// Timer/XPULSE
(*Ist x_Ein auf true, wird x_Aus auf true gesetzt mit der eingegebenen Ablaufzeit, unabhängig ob x_Ein früher abfällt,
als die eingegebene Ablaufzeit.
*)
FUNCTION_BLOCK XPULSE
(*
Versionsverlauf: 
Version		|Autor	|Bemerkung
------------------------------------------------------------------------------------------------------------ 
17.05.00	|KuzR	|erste Freigabe 
17.08.00	|LeaF	|Freigabe

*)
VAR_INPUT
	x_Ein:BOOL;//Eingang
END_VAR
VAR_INPUT PERSISTENT
	t_Abl:Timestruct := (wSecond := 5);//Eingegebene Ablaufzeit	
END_VAR
VAR_OUTPUT
	x_Aus:BOOL;//Digitaler Ausgang
	t_ET:Timestruct;//Ausgang Ablaufzeit
END_VAR	
VAR
	Ein:tp;
	t_PtZeit:TIME;
	Timestruct_to_Time:Timestruct_to_Time;
	Time_to_Timestruct: Time_to_Timestruct;	
END_VAR

//Wenn Eingang True, dann läuft eingestellte Zeit ab	
	Timestruct_to_Time(t_Ein:=t_Abl , t_Aus=>t_PtZeit );
	Ein(IN:= x_Ein, PT:= t_PtZeit, Q=> x_Aus);

//Ausgabe Ablaufzeit im timestruct
	Time_to_Timestruct(t_Ein:= Ein.ET, t_Aus=> t_ET);

END_FUNCTION_BLOCK

// Uhren/ABS_Bool
(*Anti Blockiersystem für BOOL Aktoren. Wird der Aktor während der eingestellten Zeit nicht bewegt so wird dieser für eine bestimmte Dauer eingeschalten.
*)
FUNCTION_BLOCK ABS_Bool
(*
Versionsverlauf: 
Version		|Autor	|Bemerkung
------------------------------------------------------------------------------------------------------------ 
17.06.00	|Shgb	|erste Freigabe 

*)
VAR_INPUT
	x_Ein:BOOL;//Eingang
END_VAR
VAR_INPUT PERSISTENT
	t_Einschaltzeitpunkt:timestruct := (wDayOfWeek := 1, wHour := 9) ;//Wochentag mit Uhrzeit wann der Ausgang geschalten wird
	t_Dauer:timestruct := (wMinute := 2);//Dauer des Force Zycklus
END_VAR
VAR_OUTPUT
	x_Aus:BOOL;//Ausgang
END_VAR
VAR
	TOF:TOF;
	Dauer:Timestruct_to_Time;
	x_Bewegt: BOOL;
	x_Flanke: BOOL;
END_VAR

// Einschalten jede Woche, eingestellte Zeit
	IF  Globale_Uhr.systemtimestruct.wDayOfWeek = t_Einschaltzeitpunkt.wDayOfWeek  AND
		Globale_Uhr.systemtimestruct.wHour = t_Einschaltzeitpunkt.wHour AND
		Globale_Uhr.systemtimestruct.wMinute = t_Einschaltzeitpunkt.wMinute THEN
		IF NOT x_Bewegt AND NOT x_Flanke THEN
			TOF.IN:=TRUE;
		ELSE
			x_Bewegt:=FALSE;
		END_IF
		x_Flanke:=TRUE;
	ELSE
		x_Flanke:=FALSE;
	END_IF
	
//Sobald Bewegt wurde Bit setzen
	IF x_Ein THEN
		x_Bewegt:=TRUE;
	END_IF

//Timestruct to Time
	Dauer(t_Ein:=t_Dauer);
	TOF(PT:=Dauer.t_Aus);
	TOF.IN:=FALSE;

//Ausgang setzen
	x_Aus:=x_Ein OR tof.Q;

END_FUNCTION_BLOCK

// Uhren/ABS_Int
(*Anti Blockiersystem für INT Aktoren. Der Aktor wir nach Ablauf der eingestellten Zeit auf den i_Force Wert bewegt und bleibt währen der Dauer auf diesem Wert.
*)
FUNCTION_BLOCK ABS_Int
(*
Versionsverlauf: 
Version		|Autor	|Bemerkung
------------------------------------------------------------------------------------------------------------ 
17.06.00	|Shgb	|erste Freigabe 

*)
VAR_INPUT
	i_Ein:int;//Eingang
END_VAR
VAR_INPUT PERSISTENT 
	t_Einschaltzeitpunkt:timestruct := (wDay := 7);//Zeit zwischen den einzelnen Force Zycklen
	t_Dauer:timestruct := (wMinute := 2);//Dauer des Force Zycklus
END_VAR
VAR_OUTPUT
	i_Aus:INT;//Ausgang
END_VAR
VAR
	TOF: TOF;
	Dauer: Timestruct_to_Time;
	x_Bewegt: BOOL;
	i_Speicher: INT;
	x_Flanke: BOOL;
END_VAR

// Einschalten jede Woche, eingestellte Zeit
	IF  Globale_Uhr.systemtimestruct.wDayOfWeek = t_Einschaltzeitpunkt.wDayOfWeek  AND
		Globale_Uhr.systemtimestruct.wHour = t_Einschaltzeitpunkt.wHour AND
		Globale_Uhr.systemtimestruct.wMinute = t_Einschaltzeitpunkt.wMinute THEN
		IF NOT x_Bewegt AND NOT x_Flanke THEN
			TOF.IN:=TRUE;
		ELSE
			x_Bewegt:=FALSE;
			i_Speicher:=i_Ein;
		END_IF
		x_Flanke:=TRUE;
	ELSE
		x_Flanke:=FALSE;
	END_IF
	
//Sobald Bewegt wurde Bit setzen
	IF i_Ein >= i_Speicher+10 OR i_Ein <= i_Speicher-10 THEN
		x_Bewegt:=TRUE;
	END_IF

//Timestruct to Time
	Dauer(t_Ein:=t_Dauer);
	TOF(PT:=Dauer.t_Aus);
	TOF.IN:=FALSE;

//Ausgang setzen
	IF tof.Q THEN
		i_Aus:=1000-i_Ein;	
	ELSE
		i_Aus:=i_Ein;
	END_IF;

END_FUNCTION_BLOCK

// Uhren/ABS_Real
(*Anti Blockiersystem für REAL Aktoren. Der Aktor wir nach Ablauf der eingestellten Zeit auf den f_Force Wert bewegt und bleibt währen der Dauer auf diesem Wert.
*)
FUNCTION_BLOCK ABS_Real
(*
Versionsverlauf: 
Version		|Autor	|Bemerkung
------------------------------------------------------------------------------------------------------------ 
17.06.00	|Shgb	|erste Freigabe 

*)
VAR_INPUT
	f_Ein:real;//Eingang
END_VAR
VAR_INPUT PERSISTENT 
	t_Einschaltzeitpunkt:timestruct := (wDay := 7);//Zeit zwischen den einzelnen Force Zycklen
	t_Dauer:timestruct := (wMinute := 2);//Dauer des Force Zycklus
END_VAR
VAR_OUTPUT
	f_Aus:REAL;//Ausgang
END_VAR
VAR
	TOF: TOF;
	Dauer: Timestruct_to_Time;
	x_Bewegt: BOOL;
	f_Speicher: REAL;

	x_Flanke: BOOL;
END_VAR

// Einschalten jede Woche, eingestellte Zeit
	IF  Globale_Uhr.systemtimestruct.wDayOfWeek = t_Einschaltzeitpunkt.wDayOfWeek  AND
		Globale_Uhr.systemtimestruct.wHour = t_Einschaltzeitpunkt.wHour AND
		Globale_Uhr.systemtimestruct.wMinute = t_Einschaltzeitpunkt.wMinute THEN
		IF NOT x_Bewegt AND NOT x_Flanke THEN
			TOF.IN:=TRUE;
		ELSE
			x_Bewegt:=FALSE;
			f_Speicher:=f_Ein;
		END_IF
		x_Flanke:=TRUE;
	ELSE
		x_Flanke:=FALSE;
	END_IF
	
//Sobald Bewegt wurde Bit setzen
	IF f_Ein >= f_Speicher+10 OR f_Ein <= f_Speicher-10 THEN
		x_Bewegt:=TRUE;
	END_IF

//Timestruct to Time
	Dauer(t_Ein:=t_Dauer);
	TOF(PT:=Dauer.t_Aus);
	TOF.IN:=FALSE;

//Ausgang setzen
	IF tof.Q THEN
		f_Aus:=100-f_Ein;	
	ELSE
		f_Aus:=f_Ein;
	END_IF;

END_FUNCTION_BLOCK

// Uhren/CLK_D
(*Uhr mit Tagesprogramm. Einschaltzeit => t_Ein.wHour, t_ein.wMinute und Ausschaltzeit => t_Aus.wHour und t_Aus.wMinute. Eingabe im Timestruct Format.
Vergleicht Ein- und Ausschaltzeit mit der Globalen_Uhr(Globale Variable)
*)
FUNCTION_BLOCK CLK_D
(*
Versionsverlauf: 
Version		|Autor	|Bemerkung
------------------------------------------------------------------------------------------------------------ 
17.06.00	|KuzR	|erste Freigabe 
17.08.00	|LeaF	|Freigabe

*)
VAR_INPUT Persistent
	t_Ein:timestruct;//Eingabe Einschaltzeit 
	t_Aus:timestruct;//Eingabe Ausschaltzeit 
END_VAR
VAR_OUTPUT
	x_Aus:BOOL;//Digitaler Ausgang		 
END_VAR
VAR
END_VAR

//schaltet jeden Tag ein, eingestell e Zeit  
	IF Globale_Uhr.systemtimestruct.wHour = t_Ein.wHour AND
 	   Globale_Uhr.systemtimestruct.wMinute >= t_Ein.wMinute THEN
			x_Aus:= TRUE;
	END_IF
				
//schaltet jeden Tag wieder aus, eingestellte Zeit			
	IF 	Globale_Uhr.systemtimestruct.wHour = t_Aus.wHour AND
		Globale_Uhr.systemtimestruct.wMinute >= t_Aus.wMinute THEN
			x_Aus:= FALSE;
	END_IF

END_FUNCTION_BLOCK

// Uhren/CLK_I
(*Uhr mit einem Impuls pro Tag. Einschaltzeit => t_Ein.wHour, t_ein.wMinute und Impulszeit => t_Imp.w.Second Eingabe im Timestruct Format. Vergleicht Einschaltzeit 
mit der Globalen_Uhr(Globale Variable)
*)
FUNCTION_BLOCK CLK_I
(*
Versionsverlauf: 
Version		|Autor	|Bemerkung
------------------------------------------------------------------------------------------------------------ 
17.06.00	|KuzR	|erste Freigabe 
17.08.00	|LeaF	|Freigabe

*)
VAR_INPUT Persistent
 	t_Ein:timestruct;//Eingabe Einschaltzeit 
	t_Imp:timestruct;//Eingabe Impulszeit
END_VAR
VAR_OUTPUT
	x_Aus:BOOL;//Digitaler Ausgang			 
END_VAR
VAR	
	impuls:tp;
	x_Zeit_groesser:BOOL;   
	t_ptImpuls: TIME;
	Timestruct_to_Time: Timestruct_to_Time;
END_VAR

//schaltet jeden Tag ein, eingestellte Zeit
	IF Globale_Uhr.systemtimestruct.wHour = t_Ein.wHour AND
 	   Globale_Uhr.systemtimestruct.wMinute >= t_Ein.wMinute THEN
			x_Zeit_groesser	:=TRUE;		
	ELSE
			x_Zeit_groesser :=  FALSE;
	END_IF
				
//Impulsdauer
	Timestruct_to_Time(t_Ein:=t_Imp , t_Aus=>t_ptImpuls );
	impuls(in:=x_Zeit_groesser, pt:=t_ptImpuls);
		x_Aus:= impuls.Q;
		x_Zeit_groesser:= x_Aus;

END_FUNCTION_BLOCK

// Uhren/CLK_M
(*Uhr mit Monatsprogramm. Schaltet 1mal im Monat für eine einstellbare Zeit.  Einschaltzeit => t_Ein.wDay, t_Ein.wHour, t_ein.wMinute
und Ausschaltzeit => t_Ein.wDay, t_Ein.wHour, t_ein.wMinute.
Eingabe im Timestruct Format. Vergleicht Ein- und Ausschaltzeit mit der Globalen_Uhr(Globale Variable)
*)
FUNCTION_BLOCK CLK_M
(*
Versionsverlauf: 
Version		|Autor	|Bemerkung
------------------------------------------------------------------------------------------------------------ 
17.06.00	|KuzR	|erste Freigabe 
17.08.00	|LeaF	|Freigabe

*)
VAR_INPUT Persistent
	    t_Ein:timestruct;//Eingabe Einschaltzeit 
		t_Aus:timestruct;//Eingabe Ausschaltzeit 	
END_VAR
VAR_OUTPUT
		x_Aus:BOOL;	 
END_VAR
VAR
	
		
	
	
	

		
	
	
END_VAR

// Einschalten einmal im Monat, Tag und Zeit
	IF  Globale_Uhr.systemtimestruct.wDay = t_Ein.wDay  AND
		Globale_Uhr.systemtimestruct.wHour = t_Ein.wHour AND
		Globale_Uhr.systemtimestruct.wMinute >= t_Ein.wMinute THEN
			x_Aus:= TRUE;
	END_IF
	
// Ausschalten einmal im Monat, Tag und Zeit
	IF  Globale_Uhr.systemtimestruct.wDay = t_Aus.wDay  AND
		Globale_Uhr.systemtimestruct.wHour = t_Aus.wHour AND
		Globale_Uhr.systemtimestruct.wMinute >= t_Aus.wMinute THEN
			x_Aus:= FALSE;
	END_IF

END_FUNCTION_BLOCK

// Uhren/CLK_W
(*Uhr mit Wochernprogramm. Schaltet 1 mal in der Woche für eine einstellbare Zeit.  Einschaltzeit => t_Ein.wDayofWeek, t_Ein.wHour, t_ein.wMinute
und Ausschaltzeit => t_Ein.wDayofWeek, t_Ein.wHour, t_ein.wMinute.
Eingabe im Timestruct Format. Vergleicht Ein- und Ausschaltzeit mit der Globalen_Uhr(Globale Variable)
*)
FUNCTION_BLOCK CLK_W
(*
Versionsverlauf: 
Version		|Autor	|Bemerkung
------------------------------------------------------------------------------------------------------------ 
17.06.00	|KuzR	|erste Freigabe 
17.08.00	|LeaF	|Freigabe

*)
VAR_INPUT Persistent
	t_Ein:timestruct;//Eingabe Einschaltzeit 
	t_Aus:timestruct;//Eingabe Ausschaltzeit
END_VAR
VAR_OUTPUT
	x_Aus:BOOL;//Digitaler Ausgang 
END_VAR

// Einschalten jede Woche, eingestellte Zeit
	IF  Globale_Uhr.systemtimestruct.wDayOfWeek = t_Ein.wDayOfWeek  AND
		Globale_Uhr.systemtimestruct.wHour = t_Ein.wHour AND
		Globale_Uhr.systemtimestruct.wMinute >= t_Ein.wMinute THEN
			x_Aus:= TRUE;
	END_IF
// Ausschalten, eingestellte Zeit
	IF  Globale_Uhr.systemtimestruct.wDayOfWeek = t_Aus.wDayOfWeek  AND
		Globale_Uhr.systemtimestruct.wHour = t_Aus.wHour AND
		Globale_Uhr.systemtimestruct.wMinute >= t_Aus.wMinute THEN
			x_Aus:= FALSE;
	END_IF

END_FUNCTION_BLOCK

// Uhren/CLK_W7
(*Uhr mit Wochenprogramm für jeden Wochentag. Schaltet 1 mal im Tag für eine einstellbare Zeit, jeden Wochentag einzeln wählbar.
Einschaltzeit => t_Ein.wHour, t_ein.wMinute
und Ausschaltzeit => t_Ein.wHour, t_ein.wMinute
Eingabe im Timestruct Format. Vergleicht Ein- und Ausschaltzeit mit der Globalen_Uhr(Globale Variable)
*)
FUNCTION_BLOCK CLK_W7
(*
Versionsverlauf: 
Version		|Autor	|Bemerkung
------------------------------------------------------------------------------------------------------------ 
17.06.00	|KuzR	|erste Freigabe 
17.08.00	|LeaF	|Freigabe

*)
VAR_INPUT Persistent	   	
		t_Ein_Mo:timestruct;//Eingabe Einschaltzeit Montag
		t_Aus_Mo:timestruct;//Eingabe Ausschaltzeit Montag
 		t_Ein_Di:timestruct;//Eingabe Einschaltzeit Dienstag
		t_Aus_Di:timestruct;//Eingabe Ausschaltzeit Dienstag
		t_Ein_Mi:timestruct;//Eingabe Einschaltzeit Mittwoch
		t_Aus_Mi:timestruct;//Eingabe Ausschaltzeit Mittwoch
		t_Ein_Do:timestruct;//Eingabe Einschaltzeit Donnerstag
		t_Aus_Do:timestruct;//Eingabe Ausschaltzeit Donnerstag
		t_Ein_Fr:timestruct;//Eingabe Einschaltzeit Freitag
		t_Aus_Fr:timestruct;//Eingabe Ausschaltzeit Freitag
		t_Ein_Sa:timestruct;//Eingabe Einschaltzeit Samstag
		t_Aus_Sa:timestruct;//Eingabe Ausschaltzeit Samstag
		t_Ein_So:timestruct;//Eingabe Einschaltzeit Sonntag
		t_Aus_So:timestruct;//Eingabe Ausschaltzeit Sonntag
END_VAR
VAR_OUTPUT
		x_Aus:BOOL;//Digitaler Ausgang	 
END_VAR
VAR
END_VAR

//Montag einschalten
	IF  Globale_Uhr.systemtimestruct.wDayOfWeek = 1  AND
		Globale_Uhr.systemtimestruct.wHour = t_Ein_Mo.wHour AND
		Globale_Uhr.systemtimestruct.wMinute >= t_Ein_Mo.wMinute THEN
			x_Aus:= TRUE;
			END_IF
//Montag ausschalten	
	IF  Globale_Uhr.systemtimestruct.wDayOfWeek = 1  AND
		Globale_Uhr.systemtimestruct.wHour = t_Aus_MO.wHour AND
		Globale_Uhr.systemtimestruct.wMinute >= t_Aus_MO.wMinute THEN
			x_Aus:= FALSE;
			END_IF
//Dienstag einschalten
	IF  Globale_Uhr.systemtimestruct.wDayOfWeek = 2  AND
		Globale_Uhr.systemtimestruct.wHour = t_Ein_Di.wHour AND
		Globale_Uhr.systemtimestruct.wMinute >= t_Ein_Di.wMinute THEN
			x_Aus:= TRUE;
			END_IF
//Dienstag ausschalten	
	IF  Globale_Uhr.systemtimestruct.wDayOfWeek = 2  AND
		Globale_Uhr.systemtimestruct.wHour = t_Aus_Di.wHour AND
		Globale_Uhr.systemtimestruct.wMinute >= t_Aus_Di.wMinute THEN
			x_Aus:= FALSE;
			END_IF
//Mittwoch einschalten
	IF  Globale_Uhr.systemtimestruct.wDayOfWeek = 3  AND
		Globale_Uhr.systemtimestruct.wHour = t_Ein_Mi.wHour AND
		Globale_Uhr.systemtimestruct.wMinute >= t_Ein_Mi.wMinute THEN
			x_Aus:= TRUE;
			END_IF
//Mittwoch ausschalten	
	IF  Globale_Uhr.systemtimestruct.wDayOfWeek = 3  AND
		Globale_Uhr.systemtimestruct.wHour = t_Aus_Mi.wHour AND
		Globale_Uhr.systemtimestruct.wMinute >= t_Aus_Mi.wMinute THEN
			x_Aus:= FALSE;
			END_IF		
//Donnerstag einschalten
	IF  Globale_Uhr.systemtimestruct.wDayOfWeek = 4  AND
		Globale_Uhr.systemtimestruct.wHour = t_Ein_Do.wHour AND
		Globale_Uhr.systemtimestruct.wMinute >= t_Ein_Do.wMinute THEN
			x_Aus:= TRUE;
			END_IF
//Donnerstag ausschalten	
	IF  Globale_Uhr.systemtimestruct.wDayOfWeek = 4  AND
		Globale_Uhr.systemtimestruct.wHour = t_Aus_Do.wHour AND
		Globale_Uhr.systemtimestruct.wMinute >= t_Aus_Do.wMinute THEN
			x_Aus:= FALSE;
			END_IF

//Freitag einschalten
	IF  Globale_Uhr.systemtimestruct.wDayOfWeek = 5  AND
		Globale_Uhr.systemtimestruct.wHour = t_Ein_Fr.wHour AND
		Globale_Uhr.systemtimestruct.wMinute >= t_Ein_Fr.wMinute THEN
			x_Aus:= TRUE;
			END_IF
//Freitag ausschalten	
	IF  Globale_Uhr.systemtimestruct.wDayOfWeek = 5  AND
		Globale_Uhr.systemtimestruct.wHour = t_Aus_Fr.wHour AND
		Globale_Uhr.systemtimestruct.wMinute >= t_Aus_Fr.wMinute THEN
			x_Aus:= FALSE;
			END_IF		
//Samstag einschalten
	IF  Globale_Uhr.systemtimestruct.wDayOfWeek = 6  AND
		Globale_Uhr.systemtimestruct.wHour = t_Ein_Sa.wHour AND
		Globale_Uhr.systemtimestruct.wMinute >= t_Ein_Sa.wMinute THEN
			x_Aus:= TRUE;
			END_IF
//Samstag ausschalten	
	IF  Globale_Uhr.systemtimestruct.wDayOfWeek = 6  AND
		Globale_Uhr.systemtimestruct.wHour = t_Aus_Sa.wHour AND
		Globale_Uhr.systemtimestruct.wMinute >= t_Aus_Sa.wMinute THEN
			x_Aus:= FALSE;
			END_IF	
//Sonntag einschalten
	IF  Globale_Uhr.systemtimestruct.wDayOfWeek = 0  AND
		Globale_Uhr.systemtimestruct.wHour = t_Ein_So.wHour AND
		Globale_Uhr.systemtimestruct.wMinute >= t_Ein_So.wMinute THEN
			x_Aus:= TRUE;
			END_IF
//Sonntag ausschalten	
	IF  Globale_Uhr.systemtimestruct.wDayOfWeek = 0  AND
		Globale_Uhr.systemtimestruct.wHour = t_Aus_So.wHour AND
		Globale_Uhr.systemtimestruct.wMinute >= t_Aus_So.wMinute THEN
			x_Aus:= FALSE;
			END_IF

END_FUNCTION_BLOCK

// Uhren/CLK_Y
(*Uhr mit Jahresrogramm. Schaltet 1 mal im Jahr für eine einstellbare Zeit.  Einschaltzeit => t_Ein.wMonth, t_Ein.wDay, t_Ein.wHour, t_ein.wMinute
und Ausschaltzeit => t_Aus.wMonth, t_Ein.wDay, t_Ein.wHour, t_ein.wMinute.
Eingabe im Timestruct Format. Vergleicht Ein- und Ausschaltzeit mit der Globalen_Uhr(Globale Variable)
*)
FUNCTION_BLOCK CLK_Y
(*
Versionsverlauf: 
Version		|Autor	|Bemerkung
------------------------------------------------------------------------------------------------------------ 
17.06.00	|KuzR	|erste Freigabe 
17.08.00	|LeaF	|Freigabe

*)
VAR_INPUT Persistent
	t_Ein:timestruct;//Eingabe Einschaltzeit
	t_Aus:timestruct;//Eingabe Ausschaltzeit	

END_VAR
VAR_OUTPUT
	x_Aus:BOOL;			 
END_VAR
VAR
END_VAR

// Einschalten einmal im Jahr, Zeit, Tagnummer und Monat
	IF Globale_Uhr.systemtimestruct.wMonth = t_Ein.wMonth AND
 	   Globale_Uhr.systemtimestruct.wDay = t_Ein.wDay AND
	   Globale_Uhr.systemtimestruct.wHour = t_Ein.wHour AND
	   Globale_Uhr.systemtimestruct.wMinute >= t_Ein.wMinute THEN
			x_Aus:= TRUE;		
	END_IF
			
// Ausschalten Zeit, Tagnummer und Monat 	
	IF Globale_Uhr.systemtimestruct.wMonth = t_Aus.wMonth AND
 	   Globale_Uhr.systemtimestruct.wDay = t_Aus.wDay AND
	   Globale_Uhr.systemtimestruct.wHour = t_Aus.wHour AND
	   Globale_Uhr.systemtimestruct.wMinute >= t_Aus.wMinute THEN			
			x_Aus:= FALSE;
	END_IF

END_FUNCTION_BLOCK

// Uhren/FerienPRG
(*FB Ferienprogramm, Wenn FB aktiviert und die Schaltuhr aktiv ist, schaltet die Freigabe x_BM und der Sollwert Eingang wird auf
den Ausgang geschrieben. Es muss nur die Ausschaltzeit eingegeben werden t_Aus.wMonth, => t_Aus.wDay, t_Aus.wHour, t_Aus.wMinute.
Sobald die Zeit abgelaufen ist, wird der Sollwert Ausgang auf 0 gesetzt und der Ausgang x_BM wird auf false gesetzt.
*)
FUNCTION_BLOCK FerienPRG
(*
Versionsverlauf: 
Version		|Autor	|Bemerkung
------------------------------------------------------------------------------------------------------------ 
17.07.00	|KuzR	|erste Freigabe 
17.08.00	|LeaF	|Freigabe

*)
VAR_INPUT PERSISTENT
	x_Akt:BOOL;//Aktivierung
	t_Aus:TIMESTRUCT;//Ausschaltzeit
	f_SW_fix:REAL;//Sollwert
END_VAR
VAR_OUTPUT
	x_BM:BOOL;//Freigabe
	f_SW:REAL;//Sollwert
	t_Restzeit:timestruct;//Anzeige Restzeit
END_VAR
VAR
	ein: BOOL;
	x_Aus_Uhr:BOOL;
	x_ein:BOOL;
	t_Restzeit1:TIME;
	t_Ausschalt: TIME;
	t_Global:TIME;
	CLK_M: CLK_M;
	Timestruct_to_Time: Timestruct_to_Time;
	Time_to_Timestruct: Time_to_Timestruct;
	SWITCH_REAL: SWITCH_REAL;
	
	CLK_Y: CLK_Y;
END_VAR

//Kommentar

//Monatsuhr, Zeiteingabe im Timestruct
		CLK_Y(t_Ein:= Globale_Uhr.systemtimestruct, t_Aus:=t_Aus , x_Aus=>x_Aus_Uhr );
//Freigabe schalten
 		x_BM:= x_Akt AND x_Aus_Uhr;

//Timestruct to time
		Timestruct_to_Time(t_Ein:=t_Aus , t_Aus=>t_Ausschalt );
		Timestruct_to_Time(t_Ein:=Globale_Uhr.systemtimestruct , t_Aus=>t_Global);	
			
//Restzeit berechnen im Time Format
		t_Restzeit1:=t_Ausschalt-t_Global;
	IF t_Ausschalt < t_Global THEN
		t_Restzeit1:=T#0S;
	END_IF
	
//Time to timestruct
	Time_to_Timestruct(t_Ein:= t_Restzeit1, t_Aus=> t_Restzeit);

//Sollwert in den Ausgang schreiben	
	SWITCH_REAL(x_Ein:=x_BM , f_Ein_1:=0 , f_Ein_2:=f_SW_fix , f_Aus=>f_SW );
		
	IF NOT x_Aus_Uhr THEN
		x_Akt:=FALSE;
	END_IF

END_FUNCTION_BLOCK

// Verdichter/Einsatzgrenzen_Normal
(*Überwacht die Einsatzgrenzen der Kompressoren und gibt mit einem BOOL an ob diese sich noch in den Einsatzgrenzen befinden. Ein Toleranzband kann zusätzlich mit einer Zeit bestimmt werden.
Verlässt der Kompressor die Einsatzgrenzen ober wird zu lange im Toleranzband betrieben so wird das Ausgangsbool auf FALSE gesetzt. Für weitere Infos siehe Beschrieb im FB.
*)
FUNCTION_BLOCK Einsatzgrenzen_Normal
(*
Versionsverlauf: 
Version		|Autor	|Bemerkung
------------------------------------------------------------------------------------------------------------ 
17.06.00	|Shgb	|erste Freigabe 
17.06.01	|ShgB	|von Integer auf Real geändert
17.06.02	|ShgB	|Von Time auf Timestruct geändert
17.07.00	|ShgB	|MOP Berechnung angepasst

		  F	_____________5__________ E
		  /							\ 4
	  6	/							 \ D
	  /								 | 3
  G /								 | C
	|								/  
	|							  /
  7 |							/ 2
	|_________________________/
	A			1			  B
*)
VAR_INPUT 
	f_Verd:REAL;//Aktuelle Verdampfungstemperatur
	f_Kond:REAL;//Aktuelle Kondensationstemperatur
	x_Betriebsmeldung: BOOL;//Sobald die Betriebsmeldung kommt wird die Auswertung um die eingestellte Zeit verzögert aktiv
	x_SW_Reset:BOOL;//Setzt die Standardwerte für den Kompressorty zurück
	dut_Kompressortyp:SW_Einsatzgrenzen:=SW_ALZ.Bitzer_Scroll_R410a;//Kompressortyp als DUT Angabe Standard Bitzer Scroll 410a
END_VAR
VAR_INPUT PERSISTENT
	f_MinVerd:REAL;//Minimale Verdampfungstemperatur Linie 7
	f_MaxVerd:REAL;//Maximale Verdampfungstemperatur Linie 3
	f_MinKond:REAL;//Minimale Kondensationstemperatur Punkt A
	f_MaxKond:REAL;//Maximale Kondensationstemperatur Linie 5
	f_BVerd:REAL;//Verdampfungstemperatur beim Punkt B
	f_BKond:REAL;//Kondensationstemperatur beim Punkt B
	f_CKond:REAL;//Kondensationstemperatur beim Punkt C
	f_DKond:REAL;//Kondensationstemperatur beim Punkt D
	f_EVerd:REAL;//Verdampfungstemperatur beim Punkt E
	f_FVerd:REAL;//Verdampfungstemperatur beim Punkt F
	f_GKond:REAL;//Kondensationstemperatur beim Punkt G
	f_Toleranz:REAL:=1;//Breite des Toleranzbandes in °C
	t_Toleranz:timestruct := (wMinute := 5);//Zeit die der Kompressor im Toleranzband sein darf
	f_GUI_Zoom:REAL;//Zoomfaktor für das Vergrössern der Grafik
	i_GUI_VersatzX:INT;//Versatz der Grafik in X Richtung (Verdampfung)
	i_GUI_VersatzY:INT;//Versatz der Grafik in Y Richtung (Kondensation)
END_VAR
VAR_OUTPUT
	f_ActMinKond:REAL;//Aktuelle mindest Kondensation laut Einsatzgrenzendiagramm
	f_ActMaxKond:REAL;//Aktuelle maximale Kondensation laut Einsatzgrenzendiagramm
	f_ActMinVerd:REAL;//Aktuelle mindest Verdampfung laut Einsatgrenzendiagramm
	f_ActMaxVerd:REAL;//Aktuelle maximale Verdampfung laut Einsatzgrenzendiagramm
	x_Aus:BOOL;//Befindet sich der Kompressor in den Einsatzgrenzen
	x_BM_ND:BOOL;//Kompressor befindet sich im Toleranzband auf der Niederdruckseite
	x_AL_ND:BOOL;//Kompressor ist ausserhalb der Einsatzgrenzen auf der Niederdruckseite
	x_BM_HD:BOOL;//Kompressor befindet sich im Toleranzband auf der Hochdruckseite
	x_AL_HD:BOOL;//Kompressor ist ausserhalb der Einsatzgrenzen auf der Hochdruckseite
	x_BM_MOP: BOOL;//Kompressor befindet sich im Toleranzband vor dem MOP Alarm
	x_AL_MOP: BOOL;//MOP wurde überschritten
END_VAR
VAR
	Timer: TON;
	x_Timer:BOOL;
	Maximum: Maximum;
	Linie1_Verd: Converter2Punkt;
	Linie1_Kond: Converter2Punkt;
	Linie2_Verd: Converter2Punkt;
	Linie2_Kond: Converter2Punkt;
	Linie4_Kond: Converter2Punkt;
	Linie4_Verd: Converter2Punkt;
	Linie6_Verd: Converter2Punkt;
	Linie6_Kond: Converter2Punkt;
	Minimum: Minimun;
	t_Temp: TIME;
	Timestruct_to_Time:Timestruct_to_Time;
	FB_MIN_KD: maximum;
	FB_MIN_VD: maximum;
	FB_MAX_KD: Minimun;
	FB_MAX_VD: Minimun;
	Betriebsmeldung:Ton;
END_VAR
VAR PERSISTENT
	x_Laden:BOOL;//Variable ist beim ersten aufstarten False und lädt somit die eingestellten Daten
END_VAR
VAR//Variablen für Grafik
	f_GUI_Verd:REAL;//Aktuelle Verdampfungstemperatur
	f_GUI_Kond:REAL;//Aktuelle Kondensationstemperatur
	f_GUI_MinVerd:REAL;//Minimale Verdampfungstemperatur Linie 7
	f_GUI_MaxVerd:REAL;//Maximale Verdampfungstemperatur Linie 3
	f_GUI_MinKond:REAL;//Minimale Kondensationstemperatur Punkt A
	f_GUI_MaxKond:REAL;//Maximale Kondensationstemperatur Linie 5
	f_GUI_BVerd:REAL;//Verdampfungstemperatur beim Punkt B
	f_GUI_BKond:REAL;//Kondensationstemperatur beim Punkt B
	f_GUI_CKond:REAL;//Kondensationstemperatur beim Punkt C
	f_GUI_DKond:REAL;//Kondensationstemperatur beim Punkt D
	f_GUI_EVerd:REAL;//Verdampfungstemperatur beim Punkt E
	f_GUI_FVerd:REAL;//Verdampfungstemperatur beim Punkt F
	f_GUI_GKond:REAL;//Kondensationstemperatur beim Punkt G
END_VAR

//Linienberechnungen
	//Linie 1
		Linie1_Verd(
			f_Ein:= f_Verd, 
			f_Ein_Min:= f_MinVerd, 
			f_Ein_Max:= f_BVerd, 
			f_Aus_Min:= f_MinKond, 
			f_Aus_Max:= f_BKond);
			
		Linie1_Kond(
			f_Ein:= f_Kond, 
			f_Ein_Min:= f_MinKond, 
			f_Ein_Max:= f_BKond, 
			f_Aus_Min:= f_MinVerd, 
			f_Aus_Max:= f_BVerd);
			
	//Linie 2
		Linie2_Verd(
			f_Ein:= f_Verd, 
			f_Ein_Min:= f_BVerd, 
			f_Ein_Max:= f_MaxVerd, 
			f_Aus_Min:= f_BKond, 
			f_Aus_Max:= f_CKond);
			
		Linie2_Kond(
			f_Ein:= f_Kond, 
			f_Ein_Min:= f_BVerd, 
			f_Ein_Max:= f_MaxVerd, 
			f_Aus_Min:= f_BKond, 
			f_Aus_Max:= f_CKond);
			
	//Linie 4
		Linie4_Kond(
			f_Ein:= f_Kond, 
			f_Ein_Min:= f_MaxKond, 
			f_Ein_Max:= f_DKond, 
			f_Aus_Min:= f_EVerd, 
			f_Aus_Max:= f_MaxVerd);
			
		Linie4_Verd(
			f_Ein:= f_Verd, 
			f_Ein_Min:= f_EVerd, 
			f_Ein_Max:= f_MaxVerd, 
			f_Aus_Min:= f_MaxKond, 
			f_Aus_Max:= f_DKond);
			
	//Linie 6
		Linie6_Verd(
			f_Ein:= f_Verd, 
			f_Ein_Min:= f_MinVerd, 
			f_Ein_Max:= f_FVerd, 
			f_Aus_Min:= f_GKond, 
			f_Aus_Max:= f_MaxKond);
				
		Linie6_Kond(
			f_Ein:= f_Kond, 
			f_Ein_Min:= f_GKond, 
			f_Ein_Max:= f_MaxKond, 
			f_Aus_Min:= f_MinVerd, 
			f_Aus_Max:= f_FVerd);
			
//Minimale Kondensationstemperatur wird durch die Linien 1,  2 und f_MinKond vom Einsatzgrenzendiagramm gegeben. Die höhere von beiden wird genommen.
	FB_MIN_KD(
		f_Ein1:= Linie1_Verd.f_Aus, 
		f_Ein2:= Linie2_Verd.f_Aus, 
		f_Ein3:= f_MinKond, 
		f_Aus=> f_ActMinKond);
			
//Maximale Kondensationstemperaturwird durch Linie 4, 6 und f_MaxKond vom Einsatzgrenzendiagramm gegeben. Die kleinere von den dreien wird genommen. Linie 5 ist f_MaxKond
	FB_MAX_KD(
		f_Ein1:=Linie4_Verd.f_Aus,
		f_Ein2:=Linie6_Verd.f_Aus,
		f_Ein3:=f_MaxKond,
		f_Aus=>f_ActMaxKond);
			
//Minimale Verdampfungstemperatur durch Linie 6 und f_MinVerd gegeben
	FB_MIN_VD(
		f_Ein1:=Linie6_Kond.f_Aus,
		f_Ein2:= f_MinVerd,
		f_Aus=>f_ActMinVerd);
				
//Maximale Verdampfungstemperatur 
	IF f_Kond <= f_BKond AND f_Kond>= f_MinKond THEN
		f_ActMaxVerd:=Linie1_Kond.f_Aus;
	ELSE
		FB_MAX_VD(
			f_Ein1:=Linie2_Kond.f_Aus,
			f_Ein2:=Linie4_Kond.f_Aus,
			f_Ein3:=f_MaxVerd,
			f_Aus=>f_ActMaxVerd);
	END_IF

//TImestruct to Time
	Timestruct_to_Time(t_Ein:=t_Toleranz);
	
//Auswertung ob in den Einsatzgrenzen mit Timer
	Betriebsmeldung(IN:=x_Betriebsmeldung,PT:=Timestruct_to_Time.t_Aus);

	Timer(IN:= f_Verd < f_ActMinVerd+f_Toleranz OR
		f_Verd > f_ActMaxVerd-f_Toleranz OR
		f_Kond < f_ActMinKond+f_Toleranz OR
		f_Kond > f_ActMaxKond-f_Toleranz, PT:= Timestruct_to_Time.t_Aus, Q=> x_Timer, ET=> );
			
	x_Aus :=NOT Betriebsmeldung.Q OR(f_Verd > f_ActMinVerd AND
		f_Verd < f_ActMaxVerd AND
		f_Kond > f_ActMinKond AND
		f_Kond < f_ActMaxKond AND
		NOT x_Timer);

//Alarme
	IF Globale_Variablen.x_Quittieren THEN
		x_AL_HD := FALSE;
		x_AL_ND := FALSE;
		x_AL_MOP:= FALSE;
	END_IF

	x_BM_ND:=f_Verd<f_ActMinVerd+f_Toleranz;
		
	IF f_Verd<f_ActMinVerd THEN
		x_AL_ND:=TRUE;
	END_IF
		
	x_BM_HD:=f_Kond>f_ActMaxKond-f_Toleranz;
		
	IF f_Kond>f_ActMaxKond THEN
		x_AL_HD:=TRUE;
	END_IF
	
	x_BM_MOP:=f_Verd>f_ActMaxVerd-f_Toleranz;
	
	IF f_Verd>f_ActMaxVerd THEN
		x_AL_MOP:=TRUE;
	END_IF
	
//Reset Sollwerte
	IF x_SW_Reset OR not x_Laden THEN
		f_MinVerd:=dut_Kompressortyp.f_SW_EG_MinVerd;
		f_MaxVerd:=dut_Kompressortyp.f_SW_EG_MaxVerd;
		f_MinKond:=dut_Kompressortyp.f_SW_EG_MinKond;
		f_MaxKond:=dut_Kompressortyp.f_SW_EG_MaxKond;
		f_BVerd:=dut_Kompressortyp.f_SW_EG_BVerd;
		f_BKond:=dut_Kompressortyp.f_SW_EG_BKond;
		f_CKond:=dut_Kompressortyp.f_SW_EG_CKond;
		f_DKond:=dut_Kompressortyp.f_SW_EG_DKond;
		f_EVerd:=dut_Kompressortyp.f_SW_EG_EVerd;
		f_FVerd:=dut_Kompressortyp.f_SW_EG_FVerd;
		f_GKond:=dut_Kompressortyp.f_SW_EG_GKond;
		x_Laden:=TRUE;
	END_IF
	
//GUI Anpassungen
	f_GUI_Verd:=f_Verd*f_GUI_Zoom+i_GUI_VersatzX;
	f_GUI_Kond:=f_Kond*f_GUI_Zoom+i_GUI_VersatzY*-1;
	f_GUI_MinVerd:=f_MinVerd*f_GUI_Zoom+i_GUI_VersatzX;
	f_GUI_MaxVerd:=f_MaxVerd*f_GUI_Zoom+i_GUI_VersatzX;
	f_GUI_MinKond:=f_MinKond*f_GUI_Zoom+i_GUI_VersatzY*-1;
	f_GUI_MaxKond:=f_MaxKond*f_GUI_Zoom+i_GUI_VersatzY*-1;
	f_GUI_BVerd:=f_BVerd*f_GUI_Zoom+i_GUI_VersatzX;
	f_GUI_BKond:=f_BKond*f_GUI_Zoom+i_GUI_VersatzY*-1;
	f_GUI_CKond:=f_CKond*f_GUI_Zoom+i_GUI_VersatzY*-1;
	f_GUI_DKond:=f_DKond*f_GUI_Zoom+i_GUI_VersatzY*-1;
	f_GUI_EVerd:=f_EVerd*f_GUI_Zoom+i_GUI_VersatzX;
	f_GUI_FVerd:=f_FVerd*f_GUI_Zoom+i_GUI_VersatzX;
	f_GUI_GKond:=f_GKond*f_GUI_Zoom+i_GUI_VersatzY*-1;

END_FUNCTION_BLOCK

// Verdichter/FIFO
(*Funktionsbaustein zum Abgleich der Betriebsstunden. Der Kompressor mit der geringeren Anzahl an Betriebsstunden wird als nächstes in Betrieb genommen. 
Beim Ausschalten werden die Kompressoren nach dem FIFO (First in frist out) Prinzip ausgeschalten.
*)
FUNCTION_BLOCK FIFO
(*
Versionsverlauf: 
Version		|Autor	|Bemerkung
------------------------------------------------------------------------------------------------------------ 
17.06.00	|Shgb	|erste Freigabe
17.07.00	|Shgb	|Bool zum Kompressorwechsel
17.08.00	|LeaF	|Freigabe

*)
VAR_INPUT
	i_Stufen:INT;//Anzahl der angeforderten Stufen
	x_En1:BOOL;//Betriebstunden von Kompressor 1
	t_Betriebsstunden1:timestruct;//Betriebstunden von Kompressor 1
	x_En2:BOOL;//Betriebstunden von Kompressor 2
	t_Betriebsstunden2:timestruct;//Betriebstunden von Kompressor 2
	x_En3:BOOL;//Betriebstunden von Kompressor 3
	t_Betriebsstunden3:timestruct;//Betriebstunden von Kompressor 3
	x_En4:BOOL;//Betriebstunden von Kompressor 4
	t_Betriebsstunden4:timestruct;//Betriebstunden von Kompressor 4
	x_En5:BOOL;//Betriebstunden von Kompressor 5
	t_Betriebsstunden5:timestruct;//Betriebstunden von Kompressor 5
	x_En6:BOOL;//Betriebstunden von Kompressor 6
	t_Betriebsstunden6:timestruct;//Betriebstunden von Kompressor 6
	x_En7:BOOL;//Betriebstunden von Kompressor 7
	t_Betriebsstunden7:timestruct;//Betriebstunden von Kompressor 7
	x_En8:BOOL;//Betriebstunden von Kompressor 8
	t_Betriebsstunden8:timestruct;//Betriebstunden von Kompressor 8
	x_Wechsel: BOOL;	// Befhel für die Umschaltung der betriebenen Kompressoren.
END_VAR
VAR_OUTPUT
	x_Aus1:BOOL;//Einschaltbefehl Kompressor 1
	x_Aus2:BOOL;//Einschaltbefehl Kompressor 2
	x_Aus3:BOOL;//Einschaltbefehl Kompressor 3
	x_Aus4:BOOL;//Einschaltbefehl Kompressor 4
	x_Aus5:BOOL;//Einschaltbefehl Kompressor 5
	x_Aus6:BOOL;//Einschaltbefehl Kompressor 6
	x_Aus7:BOOL;//Einschaltbefehl Kompressor 7
	x_Aus8:BOOL;//Einschaltbefehl Kompressor 8
END_VAR
VAR
	t_Ein1,t_Ein2,t_Ein3,t_Ein4:DT;
	t_Ein5,t_Ein6,t_Ein7,t_Ein8:DT;
	Count: COUNT;
	i_Count: INT;
	x_Speicher: BOOL;
	x_1_2: Timestruct_Kleiner_Gleich_Timestruct;
	x_1_3: Timestruct_Kleiner_Gleich_Timestruct;
	x_1_4: Timestruct_Kleiner_Gleich_Timestruct;
	x_1_5: Timestruct_Kleiner_Gleich_Timestruct;
	x_1_6: Timestruct_Kleiner_Gleich_Timestruct;
	x_1_7: Timestruct_Kleiner_Gleich_Timestruct;
	x_1_8: Timestruct_Kleiner_Gleich_Timestruct;
	x_2_1: Timestruct_Kleiner_Gleich_Timestruct;
	x_2_3: Timestruct_Kleiner_Gleich_Timestruct;
	x_2_4: Timestruct_Kleiner_Gleich_Timestruct;
	x_2_5: Timestruct_Kleiner_Gleich_Timestruct;
	x_2_6: Timestruct_Kleiner_Gleich_Timestruct;
	x_2_7: Timestruct_Kleiner_Gleich_Timestruct;
	x_2_8: Timestruct_Kleiner_Gleich_Timestruct;
	x_3_1: Timestruct_Kleiner_Gleich_Timestruct;
	x_3_2: Timestruct_Kleiner_Gleich_Timestruct;
	x_3_4: Timestruct_Kleiner_Gleich_Timestruct;
	x_3_5: Timestruct_Kleiner_Gleich_Timestruct;
	x_3_6: Timestruct_Kleiner_Gleich_Timestruct;
	x_3_7: Timestruct_Kleiner_Gleich_Timestruct;
	x_3_8: Timestruct_Kleiner_Gleich_Timestruct;
	x_4_1: Timestruct_Kleiner_Gleich_Timestruct;
	x_4_2: Timestruct_Kleiner_Gleich_Timestruct;
	x_4_3: Timestruct_Kleiner_Gleich_Timestruct;
	x_4_5: Timestruct_Kleiner_Gleich_Timestruct;
	x_4_6: Timestruct_Kleiner_Gleich_Timestruct;
	x_4_7: Timestruct_Kleiner_Gleich_Timestruct;
	x_4_8: Timestruct_Kleiner_Gleich_Timestruct;
	x_5_1: Timestruct_Kleiner_Gleich_Timestruct;
	x_5_2: Timestruct_Kleiner_Gleich_Timestruct;
	x_5_3: Timestruct_Kleiner_Gleich_Timestruct;
	x_5_4: Timestruct_Kleiner_Gleich_Timestruct;
	x_5_6: Timestruct_Kleiner_Gleich_Timestruct;
	x_5_7: Timestruct_Kleiner_Gleich_Timestruct;
	x_5_8: Timestruct_Kleiner_Gleich_Timestruct;
	x_6_1: Timestruct_Kleiner_Gleich_Timestruct;
	x_6_2: Timestruct_Kleiner_Gleich_Timestruct;
	x_6_3: Timestruct_Kleiner_Gleich_Timestruct;
	x_6_4: Timestruct_Kleiner_Gleich_Timestruct;
	x_6_5: Timestruct_Kleiner_Gleich_Timestruct;
	x_6_7: Timestruct_Kleiner_Gleich_Timestruct;
	x_6_8: Timestruct_Kleiner_Gleich_Timestruct;
	x_7_1: Timestruct_Kleiner_Gleich_Timestruct;
	x_7_2: Timestruct_Kleiner_Gleich_Timestruct;
	x_7_3: Timestruct_Kleiner_Gleich_Timestruct;
	x_7_4: Timestruct_Kleiner_Gleich_Timestruct;
	x_7_5: Timestruct_Kleiner_Gleich_Timestruct;
	x_7_6: Timestruct_Kleiner_Gleich_Timestruct;
	x_7_8: Timestruct_Kleiner_Gleich_Timestruct;
	x_8_1: Timestruct_Kleiner_Gleich_Timestruct;
	x_8_2: Timestruct_Kleiner_Gleich_Timestruct;
	x_8_3: Timestruct_Kleiner_Gleich_Timestruct;
	x_8_4: Timestruct_Kleiner_Gleich_Timestruct;
	x_8_5: Timestruct_Kleiner_Gleich_Timestruct;
	x_8_6: Timestruct_Kleiner_Gleich_Timestruct;
	x_8_7: Timestruct_Kleiner_Gleich_Timestruct;
END_VAR

//Verdichter zählen
	Count(
	x_Ein_1:= x_Aus1, 
	x_Ein_2:= x_Aus2, 
	x_Ein_3:= x_Aus3, 
	x_Ein_4:= x_Aus4,
	x_Ein_5:= x_Aus5,
	x_Ein_6:= x_Aus6,
	x_Ein_7:= x_Aus7,
	x_Ein_8:= x_Aus8,
	i_Aus=> i_Count);
//Betriebsstunden vergleichen
	//Vergleich zu Verdichter 1
	x_1_2(t_Ein1:=t_Betriebsstunden1, t_Ein2:= t_Betriebsstunden2);
	x_1_3(t_Ein1:=t_Betriebsstunden1, t_Ein2:= t_Betriebsstunden3);
	x_1_4(t_Ein1:=t_Betriebsstunden1, t_Ein2:= t_Betriebsstunden4);
	x_1_5(t_Ein1:=t_Betriebsstunden1, t_Ein2:= t_Betriebsstunden5);
	x_1_6(t_Ein1:=t_Betriebsstunden1, t_Ein2:= t_Betriebsstunden6);
	x_1_7(t_Ein1:=t_Betriebsstunden1, t_Ein2:= t_Betriebsstunden7);
	x_1_8(t_Ein1:=t_Betriebsstunden1, t_Ein2:= t_Betriebsstunden8);
	//Vergleich zu Verdichter 2
	x_2_1(t_Ein1:=t_Betriebsstunden2, t_Ein2:= t_Betriebsstunden1);
	x_2_3(t_Ein1:=t_Betriebsstunden2, t_Ein2:= t_Betriebsstunden3);
	x_2_4(t_Ein1:=t_Betriebsstunden2, t_Ein2:= t_Betriebsstunden4);
	x_2_5(t_Ein1:=t_Betriebsstunden2, t_Ein2:= t_Betriebsstunden5);
	x_2_6(t_Ein1:=t_Betriebsstunden2, t_Ein2:= t_Betriebsstunden6);
	x_2_7(t_Ein1:=t_Betriebsstunden2, t_Ein2:= t_Betriebsstunden7);
	x_2_8(t_Ein1:=t_Betriebsstunden2, t_Ein2:= t_Betriebsstunden8);
	//Vergleich zu Verdichter 3
	x_3_1(t_Ein1:=t_Betriebsstunden3, t_Ein2:= t_Betriebsstunden1);
	x_3_2(t_Ein1:=t_Betriebsstunden3, t_Ein2:= t_Betriebsstunden2);
	x_3_4(t_Ein1:=t_Betriebsstunden3, t_Ein2:= t_Betriebsstunden4);
	x_3_5(t_Ein1:=t_Betriebsstunden3, t_Ein2:= t_Betriebsstunden5);
	x_3_6(t_Ein1:=t_Betriebsstunden3, t_Ein2:= t_Betriebsstunden6);
	x_3_7(t_Ein1:=t_Betriebsstunden3, t_Ein2:= t_Betriebsstunden7);
	x_3_8(t_Ein1:=t_Betriebsstunden3, t_Ein2:= t_Betriebsstunden8);
	//Vergleich zu Verdichter 4
	x_4_1(t_Ein1:=t_Betriebsstunden4, t_Ein2:= t_Betriebsstunden1);
	x_4_2(t_Ein1:=t_Betriebsstunden4, t_Ein2:= t_Betriebsstunden2);
	x_4_3(t_Ein1:=t_Betriebsstunden4, t_Ein2:= t_Betriebsstunden3);
	x_4_5(t_Ein1:=t_Betriebsstunden4, t_Ein2:= t_Betriebsstunden5);
	x_4_6(t_Ein1:=t_Betriebsstunden4, t_Ein2:= t_Betriebsstunden6);
	x_4_7(t_Ein1:=t_Betriebsstunden4, t_Ein2:= t_Betriebsstunden7);
	x_4_8(t_Ein1:=t_Betriebsstunden4, t_Ein2:= t_Betriebsstunden8);
	//Vergleich zu Verdichter 5
	x_5_1(t_Ein1:=t_Betriebsstunden5, t_Ein2:= t_Betriebsstunden1);
	x_5_2(t_Ein1:=t_Betriebsstunden5, t_Ein2:= t_Betriebsstunden2);
	x_5_3(t_Ein1:=t_Betriebsstunden5, t_Ein2:= t_Betriebsstunden3);
	x_5_4(t_Ein1:=t_Betriebsstunden5, t_Ein2:= t_Betriebsstunden4);
	x_5_6(t_Ein1:=t_Betriebsstunden5, t_Ein2:= t_Betriebsstunden6);
	x_5_7(t_Ein1:=t_Betriebsstunden5, t_Ein2:= t_Betriebsstunden7);
	x_5_8(t_Ein1:=t_Betriebsstunden5, t_Ein2:= t_Betriebsstunden8);
	//Vergleich zu Verdichter 6
	x_6_1(t_Ein1:=t_Betriebsstunden6, t_Ein2:= t_Betriebsstunden1);
	x_6_2(t_Ein1:=t_Betriebsstunden6, t_Ein2:= t_Betriebsstunden2);
	x_6_3(t_Ein1:=t_Betriebsstunden6, t_Ein2:= t_Betriebsstunden3);
	x_6_4(t_Ein1:=t_Betriebsstunden6, t_Ein2:= t_Betriebsstunden4);
	x_6_5(t_Ein1:=t_Betriebsstunden6, t_Ein2:= t_Betriebsstunden5);
	x_6_7(t_Ein1:=t_Betriebsstunden6, t_Ein2:= t_Betriebsstunden7);
	x_6_8(t_Ein1:=t_Betriebsstunden6, t_Ein2:= t_Betriebsstunden8);
	//Vergleich zu Verdichter 7
	x_7_1(t_Ein1:=t_Betriebsstunden7, t_Ein2:= t_Betriebsstunden1);
	x_7_2(t_Ein1:=t_Betriebsstunden7, t_Ein2:= t_Betriebsstunden2);
	x_7_3(t_Ein1:=t_Betriebsstunden7, t_Ein2:= t_Betriebsstunden3);
	x_7_4(t_Ein1:=t_Betriebsstunden7, t_Ein2:= t_Betriebsstunden4);
	x_7_5(t_Ein1:=t_Betriebsstunden7, t_Ein2:= t_Betriebsstunden5);
	x_7_6(t_Ein1:=t_Betriebsstunden7, t_Ein2:= t_Betriebsstunden6);
	x_7_8(t_Ein1:=t_Betriebsstunden7, t_Ein2:= t_Betriebsstunden8);
	//Vergleich zu Verdichter 8
	x_8_1(t_Ein1:=t_Betriebsstunden8, t_Ein2:= t_Betriebsstunden1);
	x_8_2(t_Ein1:=t_Betriebsstunden8, t_Ein2:= t_Betriebsstunden2);
	x_8_3(t_Ein1:=t_Betriebsstunden8, t_Ein2:= t_Betriebsstunden3);
	x_8_4(t_Ein1:=t_Betriebsstunden8, t_Ein2:= t_Betriebsstunden4);
	x_8_5(t_Ein1:=t_Betriebsstunden8, t_Ein2:= t_Betriebsstunden5);
	x_8_6(t_Ein1:=t_Betriebsstunden8, t_Ein2:= t_Betriebsstunden6);
	x_8_7(t_Ein1:=t_Betriebsstunden8, t_Ein2:= t_Betriebsstunden7);
	
//Verdichterumschaltung für einen Zyklus einen Verdichter mehr anfordern Umschaltung verläuft also quasi nahtlos
	IF x_Wechsel AND NOT x_Speicher THEN
		i_Stufen:= i_Stufen+1;
	END_IF
	x_Speicher:=x_Wechsel;
	
//Einschalten
	//Einschalten Verdichter 1
		IF x_En1 AND i_Stufen > i_Count AND NOT x_Aus1 AND
			(x_1_2.x_Aus AND x_En2 OR x_Aus2 OR NOT x_En2) AND
			(x_1_3.x_Aus AND x_En3 OR x_Aus3 OR NOT x_En3) AND
			(x_1_4.x_Aus AND x_En4 OR x_Aus4 OR NOT x_En4) AND
			(x_1_5.x_Aus AND x_En5 OR x_Aus5 OR NOT x_En5) AND
			(x_1_6.x_Aus AND x_En6 OR x_Aus6 OR NOT x_En6) AND
			(x_1_7.x_Aus AND x_En7 OR x_Aus7 OR NOT x_En7) AND
			(x_1_8.x_Aus AND x_En8 OR x_Aus8 OR NOT x_En8) THEN
			x_Aus1:=TRUE;
			t_Ein1:=Globale_Uhr.systemDateAndTime;
			i_Count:=i_Count+1;
		END_IF
	
	//Einschalten Verdichter 2
		IF x_En2 AND i_Stufen > i_Count AND NOT x_Aus2 AND
			(x_2_1.x_Aus AND x_En1 OR x_Aus1 OR NOT x_En1) AND
			(x_2_3.x_Aus AND x_En3 OR x_Aus3 OR NOT x_En3) AND
			(x_2_4.x_Aus AND x_En4 OR x_Aus4 OR NOT x_En4) AND
			(x_2_5.x_Aus AND x_En5 OR x_Aus5 OR NOT x_En5) AND
			(x_2_6.x_Aus AND x_En6 OR x_Aus6 OR NOT x_En6) AND
			(x_2_7.x_Aus AND x_En7 OR x_Aus7 OR NOT x_En7) AND
			(x_2_8.x_Aus AND x_En8 OR x_Aus8 OR NOT x_En8) THEN
			x_Aus2:=TRUE;
			t_Ein2:=Globale_Uhr.systemDateAndTime;
			i_Count:=i_Count+1;
		END_IF	
	
	//Einschalten Verdichter 3
		IF x_En3 AND i_Stufen > i_Count AND NOT x_Aus3 AND
			(x_3_1.x_Aus AND x_En1 OR x_Aus1 OR NOT x_En1) AND
			(x_3_2.x_Aus AND x_En2 OR x_Aus2 OR NOT x_En2) AND
			(x_3_4.x_Aus AND x_En4 OR x_Aus4 OR NOT x_En4) AND
			(x_3_5.x_Aus AND x_En5 OR x_Aus5 OR NOT x_En5) AND
			(x_3_6.x_Aus AND x_En6 OR x_Aus6 OR NOT x_En6) AND
			(x_3_7.x_Aus AND x_En7 OR x_Aus7 OR NOT x_En7) AND
			(x_3_8.x_Aus AND x_En8 OR x_Aus8 OR NOT x_En8) THEN
			x_Aus3:=TRUE;
			t_Ein3:=Globale_Uhr.systemDateAndTime;
			i_Count:=i_Count+1;
		END_IF	
	
	//Einschalten Verdichter 4
		IF x_En4 AND i_Stufen > i_Count AND NOT x_Aus4 AND 
			(x_4_1.x_Aus AND x_En1 OR x_Aus1 OR NOT x_En1) AND
			(x_4_2.x_Aus AND x_En2 OR x_Aus2 OR NOT x_En2) AND
			(x_4_3.x_Aus AND x_En3 OR x_Aus3 OR NOT x_En3) AND
			(x_4_5.x_Aus AND x_En5 OR x_Aus5 OR NOT x_En5) AND
			(x_4_6.x_Aus AND x_En6 OR x_Aus6 OR NOT x_En6) AND
			(x_4_7.x_Aus AND x_En7 OR x_Aus7 OR NOT x_En7) AND
			(x_4_8.x_Aus AND x_En8 OR x_Aus8 OR NOT x_En8) THEN
			x_Aus4:=TRUE;
			t_Ein4:=Globale_Uhr.systemDateAndTime;
			i_Count:=i_Count+1;
		END_IF	
	//Einschalten Verdichter 5
		IF x_En5 AND i_Stufen > i_Count AND NOT x_Aus5 AND
			(x_5_1.x_Aus AND x_En1 OR x_Aus1 OR NOT x_En1) AND
			(x_5_2.x_Aus AND x_En2 OR x_Aus2 OR NOT x_En2) AND
			(x_5_3.x_Aus AND x_En3 OR x_Aus3 OR NOT x_En3) AND
			(x_5_4.x_Aus AND x_En4 OR x_Aus4 OR NOT x_En4) AND
			(x_5_6.x_Aus AND x_En6 OR x_Aus6 OR NOT x_En6) AND
			(x_5_7.x_Aus AND x_En7 OR x_Aus7 OR NOT x_En7) AND
			(x_5_8.x_Aus AND x_En8 OR x_Aus8 OR NOT x_En8) THEN
			x_Aus5:=TRUE;
			t_Ein5:=Globale_Uhr.systemDateAndTime;
			i_Count:=i_Count+1;
		END_IF
	
	//Einschalten Verdichter 6
		IF x_En6 AND i_Stufen > i_Count AND NOT x_Aus6 AND
			(x_6_1.x_Aus AND x_En1 OR x_Aus1 OR NOT x_En1) AND
			(x_6_2.x_Aus AND x_En2 OR x_Aus2 OR NOT x_En2) AND
			(x_6_3.x_Aus AND x_En3 OR x_Aus3 OR NOT x_En3) AND
			(x_6_4.x_Aus AND x_En4 OR x_Aus4 OR NOT x_En4) AND
			(x_6_5.x_Aus AND x_En5 OR x_Aus5 OR NOT x_En5) AND
			(x_6_7.x_Aus AND x_En7 OR x_Aus7 OR NOT x_En7) AND
			(x_6_8.x_Aus AND x_En8 OR x_Aus8 OR NOT x_En8) THEN
			x_Aus6:=TRUE;
			t_Ein6:=Globale_Uhr.systemDateAndTime;
			i_Count:=i_Count+1;
		END_IF	
	
	//Einschalten Verdichter 7
		IF x_En7 AND i_Stufen > i_Count AND NOT x_Aus7 AND
			(x_7_1.x_Aus AND x_En1 OR x_Aus1 OR NOT x_En1) AND
			(x_7_2.x_Aus AND x_En2 OR x_Aus2 OR NOT x_En2) AND
			(x_7_3.x_Aus AND x_En3 OR x_Aus3 OR NOT x_En3) AND
			(x_7_4.x_Aus AND x_En4 OR x_Aus4 OR NOT x_En4) AND
			(x_7_5.x_Aus AND x_En5 OR x_Aus5 OR NOT x_En5) AND
			(x_7_6.x_Aus AND x_En6 OR x_Aus6 OR NOT x_En6) AND
			(x_7_8.x_Aus AND x_En8 OR x_Aus8 OR NOT x_En8) THEN
			x_Aus7:=TRUE;
			t_Ein7:=Globale_Uhr.systemDateAndTime;
			i_Count:=i_Count+1;
		END_IF	
	
	//Einschalten Verdichter 8
		IF x_En8 AND i_Stufen > i_Count AND NOT x_Aus8 AND
			(x_8_1.x_Aus AND x_En1 OR x_Aus1 OR NOT x_En1) AND
			(x_8_2.x_Aus AND x_En2 OR x_Aus2 OR NOT x_En2) AND
			(x_8_3.x_Aus AND x_En3 OR x_Aus3 OR NOT x_En3) AND
			(x_8_4.x_Aus AND x_En4 OR x_Aus4 OR NOT x_En4) AND
			(x_8_5.x_Aus AND x_En5 OR x_Aus5 OR NOT x_En5) AND
			(x_8_6.x_Aus AND x_En6 OR x_Aus6 OR NOT x_En6) AND
			(x_8_7.x_Aus AND x_En7 OR x_Aus7 OR NOT x_En7) THEN
			x_Aus8:=TRUE;
			t_Ein8:=Globale_Uhr.systemDateAndTime;
			i_Count:=i_Count+1;
		END_IF	
	
//Ausschalten
	//Ausschalten Verdichter 1
		IF NOT x_En1 AND x_Aus1 OR (i_Stufen < i_Count AND x_Aus1 AND
			//(t_Ein1 <= t_Ein1 OR NOT x_Aus1) AND
			(t_Ein1 <= t_Ein2 OR NOT x_Aus2) AND
			(t_Ein1 <= t_Ein3 OR NOT x_Aus3) AND
			(t_Ein1 <= t_Ein4 OR NOT x_Aus4) AND
			(t_Ein1 <= t_Ein5 OR NOT x_Aus5) AND
			(t_Ein1 <= t_Ein6 OR NOT x_Aus6) AND
			(t_Ein1 <= t_Ein7 OR NOT x_Aus7) AND
			(t_Ein1 <= t_Ein8 OR NOT x_Aus8)) THEN
			x_Aus1:=FALSE;
			i_Count:= i_Count-1;
		END_IF	
		
	//Ausschalten Verdichter 2
		IF NOT x_En2 AND x_Aus2 OR (i_Stufen < i_Count AND x_Aus2 AND
			(t_Ein2 <= t_Ein1 OR NOT x_Aus1) AND
			//(t_Ein2 <= t_Ein2 OR NOT x_Aus2) AND
			(t_Ein2 <= t_Ein3 OR NOT x_Aus3) AND
			(t_Ein2 <= t_Ein4 OR NOT x_Aus4) AND
			(t_Ein2 <= t_Ein5 OR NOT x_Aus5) AND
			(t_Ein2 <= t_Ein6 OR NOT x_Aus6) AND
			(t_Ein2 <= t_Ein7 OR NOT x_Aus7) AND
			(t_Ein2 <= t_Ein8 OR NOT x_Aus8)) THEN
			x_Aus2:=FALSE;
			i_Count:= i_Count-1;
		END_IF	
		
	//Ausschalten Verdichter 3
		IF NOT x_En3 AND x_Aus3 OR (i_Stufen < i_Count AND x_Aus3 AND
			(t_Ein3 <= t_Ein1 OR NOT x_Aus1) AND
			(t_Ein3 <= t_Ein2 OR NOT x_Aus2) AND
			//(t_Ein3 <= t_Ein3 OR NOT x_Aus3) AND
			(t_Ein3 <= t_Ein4 OR NOT x_Aus4) AND
			(t_Ein3 <= t_Ein5 OR NOT x_Aus5) AND
			(t_Ein3 <= t_Ein6 OR NOT x_Aus6) AND
			(t_Ein3 <= t_Ein7 OR NOT x_Aus7) AND
			(t_Ein3 <= t_Ein8 OR NOT x_Aus8)) THEN
			x_Aus3:=FALSE;
			i_Count:= i_Count-1;
		END_IF	
		
	//Ausschalten Verdichter 4
		IF NOT x_En4 AND x_Aus4 OR (i_Stufen < i_Count AND x_Aus4 AND
			(t_Ein4 <= t_Ein1 OR NOT x_Aus1) AND
			(t_Ein4 <= t_Ein2 OR NOT x_Aus2) AND
			(t_Ein4 <= t_Ein3 OR NOT x_Aus3) AND
			//(t_Ein4 <= t_Ein4 OR NOT x_Aus4) AND
			(t_Ein4 <= t_Ein5 OR NOT x_Aus5) AND
			(t_Ein4 <= t_Ein6 OR NOT x_Aus6) AND
			(t_Ein4 <= t_Ein7 OR NOT x_Aus7) AND
			(t_Ein4 <= t_Ein8 OR NOT x_Aus8)) THEN
			x_Aus4:=FALSE;
			i_Count:= i_Count-1;
		END_IF	
		
	//Ausschalten Verdichter 5
		IF NOT x_En5 AND x_Aus5 OR (i_Stufen < i_Count AND x_Aus5 AND
			(t_Ein5 <= t_Ein1 OR NOT x_Aus1) AND
			(t_Ein5 <= t_Ein2 OR NOT x_Aus2) AND
			(t_Ein5 <= t_Ein3 OR NOT x_Aus3) AND
			(t_Ein5 <= t_Ein4 OR NOT x_Aus4) AND
			//(t_Ein5 <= t_Ein5 OR NOT x_Aus5) AND
			(t_Ein5 <= t_Ein6 OR NOT x_Aus6) AND
			(t_Ein5 <= t_Ein7 OR NOT x_Aus7) AND
			(t_Ein5 <= t_Ein8 OR NOT x_Aus8)) THEN
			x_Aus5:=FALSE;
			i_Count:= i_Count-1;
		END_IF		
		
	//Ausschalten Verdichter 6
		IF NOT x_En6 AND x_Aus6 OR (i_Stufen < i_Count AND x_Aus6 AND
			(t_Ein6 <= t_Ein1 OR NOT x_Aus1) AND
			(t_Ein6 <= t_Ein2 OR NOT x_Aus2) AND
			(t_Ein6 <= t_Ein3 OR NOT x_Aus3) AND
			(t_Ein6 <= t_Ein4 OR NOT x_Aus4) AND
			(t_Ein6 <= t_Ein5 OR NOT x_Aus5) AND
			//(t_Ein6 <= t_Ein6 OR NOT x_Aus6) AND
			(t_Ein6 <= t_Ein7 OR NOT x_Aus7) AND
			(t_Ein6 <= t_Ein8 OR NOT x_Aus8)) THEN
			x_Aus6:=FALSE;
			i_Count:= i_Count-1;
		END_IF	
		
	//Ausschalten Verdichter 7
		IF NOT x_En7 AND x_Aus7 OR (i_Stufen < i_Count AND x_Aus7 AND
			(t_Ein7 <= t_Ein1 OR NOT x_Aus1) AND
			(t_Ein7 <= t_Ein2 OR NOT x_Aus2) AND
			(t_Ein7 <= t_Ein3 OR NOT x_Aus3) AND
			(t_Ein7 <= t_Ein4 OR NOT x_Aus4) AND
			(t_Ein7 <= t_Ein5 OR NOT x_Aus5) AND
			(t_Ein7 <= t_Ein6 OR NOT x_Aus6) AND
			//(t_Ein7 <= t_Ein7 OR NOT x_Aus7) AND
			(t_Ein7 <= t_Ein8 OR NOT x_Aus8)) THEN
			x_Aus7:=FALSE;
			i_Count:= i_Count-1;
		END_IF	
		
	//Ausschalten Verdichter 8
		IF NOT x_En8 AND x_Aus8 OR (i_Stufen < i_Count AND x_Aus8 AND
			(t_Ein8 <= t_Ein1 OR NOT x_Aus1) AND
			(t_Ein8 <= t_Ein2 OR NOT x_Aus2) AND
			(t_Ein8 <= t_Ein3 OR NOT x_Aus3) AND
			(t_Ein8 <= t_Ein4 OR NOT x_Aus4) AND
			(t_Ein8 <= t_Ein5 OR NOT x_Aus5) AND
			(t_Ein8 <= t_Ein6 OR NOT x_Aus6) AND
			(t_Ein8 <= t_Ein7 OR NOT x_Aus7) (*AND
			(t_Ein8 <= t_Ein8 OR NOT x_Aus8) *))THEN
			x_Aus8:=FALSE;
			i_Count:= i_Count-1;
		END_IF

END_FUNCTION_BLOCK

// Verdichter/Verdichter
(*Funktionsbaustein für einen Scrollverdichter mit Sanftanlauf. 
*)
FUNCTION_BLOCK Verdichter
(*
Versionsverlauf: 
Version		|Autor	|Bemerkung
------------------------------------------------------------------------------------------------------------ 
17.09.00	|Shgb	|erste Freigabe


*)
VAR_INPUT
	x_Einschaltbefehl:BOOL;//Einschaltbefehl für den Verdichter
	x_FG_Ext:BOOL:=TRUE;//Externe Freigabe
	x_RM_HD_Pressostat :BOOL;//Rückmeldung des Hochdruckpressostates
	x_RM_Sanftanlauf:BOOL;//Rückmeldung vom Sanfanlauf als Betriebsmeldung
	x_RM_Wicklungsschutz:BOOL;//Rückmeldung des Wicklungsschutzes
	x_ResetWiedereinschaltsperre:BOOL;//Wiedereinschaltsprerre quittieren
	x_ResetBetriebsstunden:BOOL;//Betriebsstunden zurücksetzen
	f_MP_ND:REAL;//Druck auf der Niederdruckseite
	f_MP_Oel:REAL;//Öldruck
	f_MT_HG:REAL;//Heissgastemperatur
END_VAR
VAR_INPUT PERSISTENT
	x_SoftSchalter:BOOL;//Handschaltung für Visu
	t_StartBetriebsstunden:Timestruct;//Betriebsstunden die beim Reset geschrieben werden
	i_StartEinschaltungen:INT;//Impulse die beim Reset geschrieben werden
	dut_Verdichtertyp:SW_Einsatzgrenzen:=SW_ALZ.Bitzer_Scroll_R410a;//Kompressortyp als DUT Angabe Standard Bitzer Scroll 410a
END_VAR
VAR_OUTPUT
	x_Freigabe:BOOL;//Verdicheter ist Freigegeben
	x_EB_TW1_Verdichter:BOOL;//Einschaltbefehl für den Verdichter Teilwicklung 1
	x_EB_TW2_Verdichter:BOOL;//Einschaltbefehl für den Verdichter Teilwicklung 2
	f_DP_Oel:REAL;//Aktuelle Oeldruckdifferenz
	t_RestzeitWiedereinschaltsperre:timestruct;//Restzeit der Wiedereinschaltsperre
	t_Betriebsstunden:timestruct;//Betriebsstunden des Kompressors
	i_Einschaltungen:INT;//Einschaltimpulse des Kompressors
	x_Reset_Wicklungsschutz:Bool;//Wicklungsschutz wird Stromlos gemacht
	x_ALS:BOOL;//Sammelalarm
	x_AL_HD_Pressostat:BOOL;//Alarm keine Rückmeldung durch Hochdruckpressostat
	x_AL_Sanftanlauf:BOOL;//Alarm keine Betriebsmeldung durch Sanftanlauf
	x_AL_Wicklungsschutz:BOOL;//Alarm Wicklungsschutz ausgelöst
	x_AL_Heissgas:BOOL;//Heissgastemperatur zu hoch
	x_AL_Oeldruck:BOOL;//Oeldruckdifferenz zu klein
END_VAR
VAR
	Betriebsstunden: Work;
	Wiedereinschaltsperre: TOF_Reset;
	Alarm_0: Alarm;
	Sanftanlauf: TON;
	Heissgass: REG2_HEIZEN;
	F_TRIG_0: F_TRIG;
	Oeldruck: REG2_HEIZEN;
	OeldruckTimer: TON;
	Teilwicklung: TON;
END_VAR
VAR // added by the converter: edge detectors and wires of the graphical bodies
    _w1 : BOOL;
END_VAR

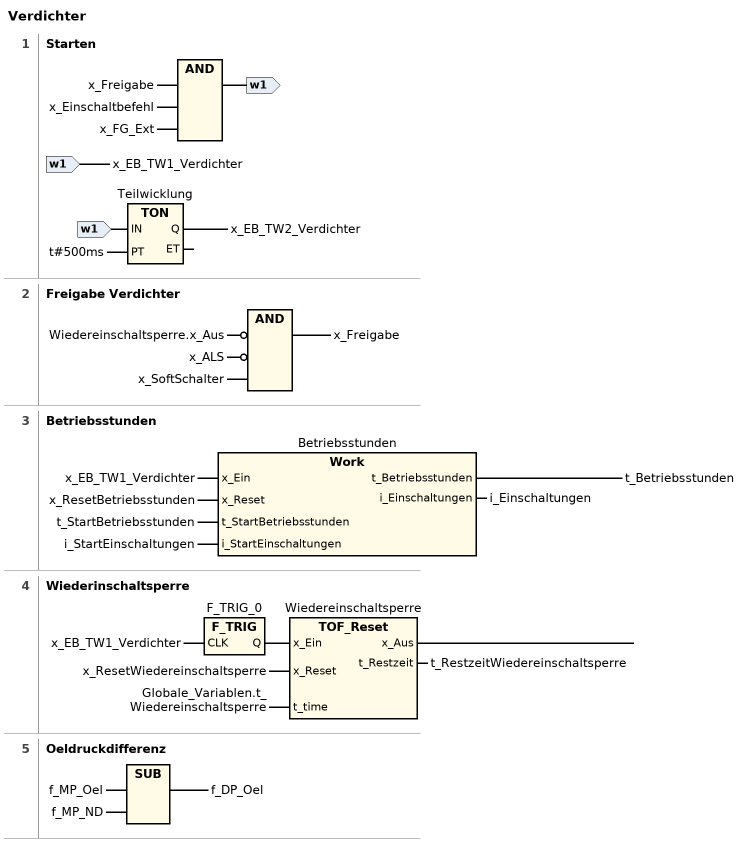
// NETWORK 1: Starten
_w1 := x_Freigabe AND x_Einschaltbefehl AND x_FG_Ext;
x_EB_TW1_Verdichter := _w1;
Teilwicklung(IN := _w1, PT := t#500ms); // TON
x_EB_TW2_Verdichter := Teilwicklung.Q;

// NETWORK 2: Freigabe Verdichter
x_Freigabe := NOT Wiedereinschaltsperre.x_Aus AND NOT x_ALS AND x_SoftSchalter;

// NETWORK 3: Betriebsstunden
Betriebsstunden(
    x_Ein := x_EB_TW1_Verdichter,
    x_Reset := x_ResetBetriebsstunden,
    t_StartBetriebsstunden := t_StartBetriebsstunden,
    i_StartEinschaltungen := i_StartEinschaltungen,
    i_Einschaltungen => i_Einschaltungen); // Work
t_Betriebsstunden := Betriebsstunden.t_Betriebsstunden;

// NETWORK 4: Wiederinschaltsperre
F_TRIG_0(CLK := x_EB_TW1_Verdichter); // F_TRIG
Wiedereinschaltsperre(
    x_Ein := F_TRIG_0.Q,
    x_Reset := x_ResetWiedereinschaltsperre,
    t_time := Globale_Variablen.t_Wiedereinschaltsperre,
    t_Restzeit => t_RestzeitWiedereinschaltsperre); // TOF_Reset

// NETWORK 5: Oeldruckdifferenz
f_DP_Oel := f_MP_Oel - f_MP_ND;

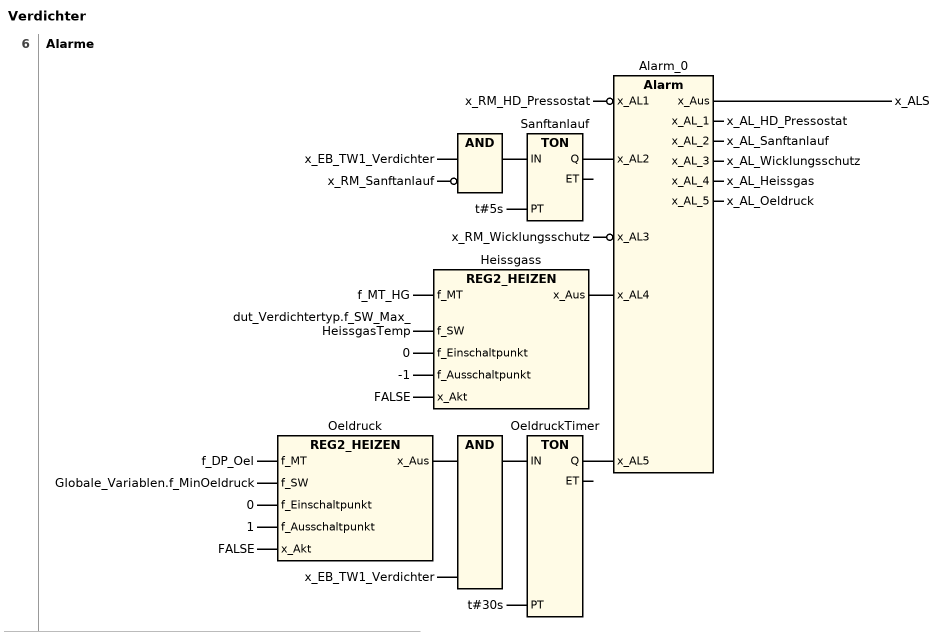
// NETWORK 6: Alarme
Sanftanlauf(IN := x_EB_TW1_Verdichter AND NOT x_RM_Sanftanlauf, PT := t#5s); // TON
Heissgass(
    f_MT := f_MT_HG,
    f_SW := dut_Verdichtertyp.f_SW_Max_HeissgasTemp,
    f_Einschaltpunkt := 0,
    f_Ausschaltpunkt := -1,
    x_Akt := FALSE); // REG2_HEIZEN
Oeldruck(
    f_MT := f_DP_Oel,
    f_SW := Globale_Variablen.f_MinOeldruck,
    f_Einschaltpunkt := 0,
    f_Ausschaltpunkt := 1,
    x_Akt := FALSE); // REG2_HEIZEN
OeldruckTimer(IN := Oeldruck.x_Aus AND x_EB_TW1_Verdichter, PT := t#30s); // TON
Alarm_0(
    x_AL1 := NOT x_RM_HD_Pressostat,
    x_AL2 := Sanftanlauf.Q,
    x_AL3 := NOT x_RM_Wicklungsschutz,
    x_AL4 := Heissgass.x_Aus,
    x_AL5 := OeldruckTimer.Q,
    x_AL_1 => x_AL_HD_Pressostat,
    x_AL_2 => x_AL_Sanftanlauf,
    x_AL_3 => x_AL_Wicklungsschutz,
    x_AL_4 => x_AL_Heissgas,
    x_AL_5 => x_AL_Oeldruck); // Alarm
x_ALS := Alarm_0.x_Aus;

END_FUNCTION_BLOCK

// Verdichter/SA_Scroll
(*Funktionsbaustein für einen Scrollverdichter mit Sanftanlauf. 
*)
FUNCTION_BLOCK SA_Scroll
(*
Versionsverlauf: 
Version		|Autor	|Bemerkung
------------------------------------------------------------------------------------------------------------ 
17.06.00	|Shgb	|erste Freigabe 
17.08.00	|LeaF	|Freigabe

*)
VAR_INPUT 
	x_HD_Pressostat :BOOL;//Rückmeldung des Hochdruckpressostates
	x_RM_Sanftanlauf:BOOL;//Rückmeldung vom Sanfanlauf als Betriebsmeldung
	x_Einschaltbefehl:BOOL;//Einschaltbefehl für den Kompressor
	x_ResetWiedereinschaltsperre:BOOL;//Wiedereinschaltsprerre quittieren
	x_ResetBetriebsstunden:BOOL;//Betriebsstunden zurücksetzen
	x_FG_Ext:BOOL:=TRUE;//Externe Freigabe
END_VAR
VAR_INPUT PERSISTENT
	x_SoftSchalter:BOOL;//Handschaltung für Visu
	t_Wiedereinschaltsperre:timestruct := (wMinute := 15);	//Sollzeit für die Wiedereinschaltsperre
	t_StartBetriebsstunden:Timestruct;//Betriebsstunden die beim Reset geschrieben werden
	i_StartEinschaltungen:INT;//Impulse die beim Reset geschrieben werden
END_VAR
VAR_OUTPUT
	x_Freigabe:BOOL;//Kompressor ist Freigegeben
	t_RestzeitWiedereinschaltsperre:timestruct;//Restzeit der Wiedereinschaltsperre
	t_Betriebsstunden:timestruct;//Betriebsstunden des Kompressors
	i_Einschaltungen:INT;//Einschaltimpulse des Kompressors
	x_Kompressor:BOOL;//Einschaltbefehl für den Kompressor
	x_AL_Sanftanlauf:BOOL;//Alarm keine Betriebsmeldung durch Sanftanlauf
	x_AL_HD_Pressostat:BOOL;//Alarm keine Rückmeldung durch Hochdruckpressostat
END_VAR
VAR
	x_Wiedereinschaltsperre,x_Alarme,x_Temp: BOOL;
	Wiedereinschaltsperre: TOF_Reset;
	TON_Sanftanlauf: TON;
	Work: Work;
	x_Speicher: BOOL;
END_VAR

//Alarme
	//Alle Alarme müssen vor dem zyklischen Ablauf geprüft werden.
	//Quittieren
	IF Globale_Variablen.x_Quittieren THEN
		x_AL_HD_Pressostat:=FALSE;
		x_AL_Sanftanlauf:=FALSE;
	END_IF
	
	//Hochdruckpressostat
	IF NOT x_HD_Pressostat THEN
		x_AL_HD_Pressostat:= TRUE;
	END_IF
	
	//Rückmeldung Sanftanlauf
	TON_Sanftanlauf(IN:=x_Kompressor AND NOT x_RM_Sanftanlauf, PT:= T#1S, Q=> x_Temp, ET=> );
	IF x_Temp THEN
		x_AL_Sanftanlauf:= TRUE;	
	END_IF
	
	x_Alarme:=x_AL_Sanftanlauf OR x_AL_HD_Pressostat;
	
//Verdichterfreigabe 
	x_Freigabe := x_SoftSchalter AND x_FG_Ext AND NOT x_Wiedereinschaltsperre AND NOT x_Alarme;
	
//Wiedereinschaltsperre
	Wiedereinschaltsperre(
		x_Ein:= NOT x_Kompressor AND x_Speicher, 
		x_Reset:= x_ResetWiedereinschaltsperre, 
		t_time:= t_Wiedereinschaltsperre, 
		x_Aus=> x_Wiedereinschaltsperre, 
		t_Restzeit=> t_RestzeitWiedereinschaltsperre);
	x_Speicher:=x_Kompressor;
		
//Einschaltbefehl
	x_Kompressor:= x_Einschaltbefehl AND x_Freigabe;
	
//Betriebsstunden
	Work(x_Ein:= x_Kompressor,
		x_Reset:= x_ResetBetriebsstunden,
		t_StartBetriebsstunden:=t_StartBetriebsstunden,
		i_StartEinschaltungen:=i_StartEinschaltungen,
		t_Betriebsstunden=> t_Betriebsstunden, 
		i_Einschaltungen=> i_Einschaltungen);

END_FUNCTION_BLOCK

// ZY_Visu/Alarmliste/Alarmliste
VISUALIZATION Alarmliste  // 800x430
END_VISUALIZATION

// ZY_Visu/Anlageseite_6/Kaeltekreis6_1
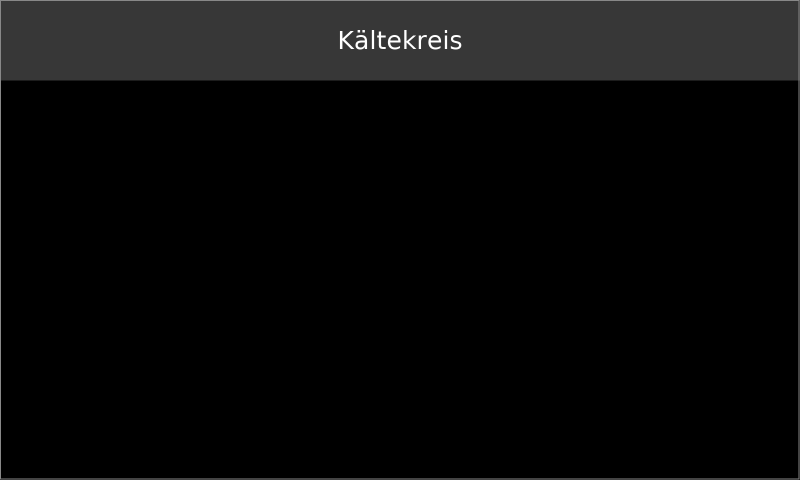
VISUALIZATION Kaeltekreis6_1  // 800x480
    Rectangle (0,0 800x80), "Kältekreis"
END_VISUALIZATION

// ZY_Visu/Anlageseite_6/Sollwertaenderung_C_6_3
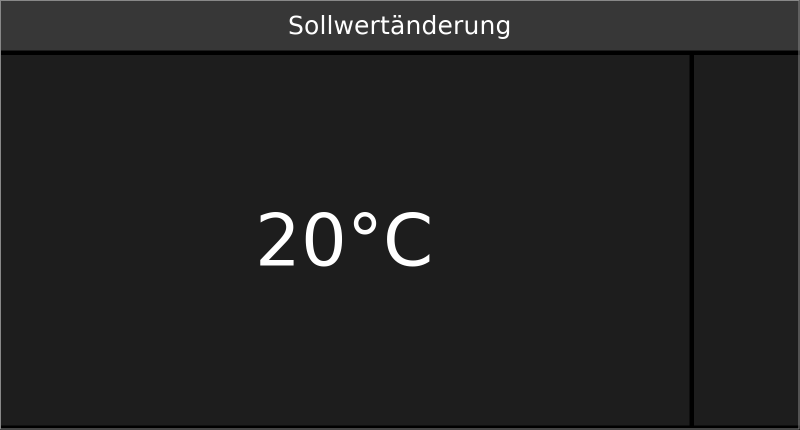
VISUALIZATION Sollwertaenderung_C_6_3  // 800x430
    Rectangle (0,0 800x50), "Sollwertänderung"
    Rectangle (0,55 689x370), "20°C"
    Rectangle (694,55 106x370)
END_VISUALIZATION

// ZY_Visu/Anlageseite_6/Zustandsanzeige
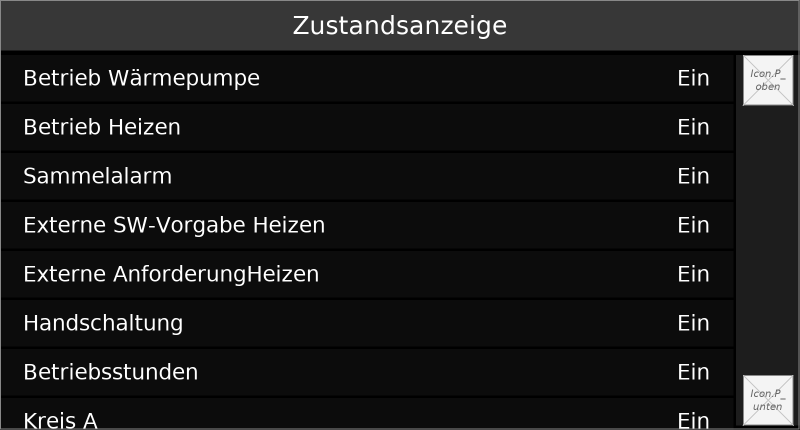
VISUALIZATION Zustandsanzeige  // 800x430
VAR_IN_OUT
	auf:BOOL;
		
END_VAR
    Image (1113,281 30x116), image: Icon.waermetauscher
    Group (0,0 800x640)
        Rectangle (0,0 800x50), "Zustandsanzeige"
        Group (0,430 800x50)
            Rectangle (0,0 800x50)
            Image (25,0 50x50), image: Icon.home
            Image (425,0 50x50), image: Icon.reinnavigieren
            Image (625,0 50x50), image: Icon.warnung_rot
            Image (125,0 50x50), image: Icon.zurueck
            Image (325,0 50x50), image: Icon.reinnavigieren
            Image (325,0 50x50), image: Icon.p_links
            Image (425,0 50x50), image: Icon.P_rechts
        Rectangle (0,55 733x46)
        Label (20,55 479x46), "Betrieb Wärmepumpe"
        Rectangle (0,104 733x46)
        Label (20,104 479x46), "Betrieb Heizen"
        Rectangle (0,153 733x46)
        Label (20,153 479x46), "Sammelalarm"
        Rectangle (0,202 733x46)
        Label (20,202 479x46), "Externe SW-Vorgabe Heizen"
        Rectangle (0,251 733x46)
        Label (20,251 479x46), "Externe AnforderungHeizen"
        Rectangle (0,300 733x46)
        Label (20,300 479x46), "Handschaltung"
        Rectangle (0,349 733x46)
        Label (20,349 479x46), "Betriebsstunden"
        Rectangle (583,55 130x46), "Ein"
        Rectangle (583,104 130x46), "Ein"
        Rectangle (0,398 733x46)
        Label (20,398 479x46), "Kreis A"
        Rectangle (0,447 733x46)
        Label (20,447 479x46), "Kreis B"
        Rectangle (0,496 733x46)
        Label (20,496 479x46), "Stufe 1"
        Rectangle (0,545 733x46)
        Label (20,545 479x46), "Stufe 2"
        Rectangle (583,545 130x46), "Ein"
        Rectangle (0,594 733x46)
        Label (20,594 479x46), "Stufe 3"
        Rectangle (583,153 130x46), "Ein"
        Rectangle (583,202 130x46), "Ein"
        Rectangle (583,251 130x46), "Ein"
        Rectangle (583,349 130x46), "Ein"
        Rectangle (583,300 130x46), "Ein"
        Rectangle (583,398 130x46), "Ein"
        Rectangle (583,447 130x46), "Ein"
        Rectangle (583,496 130x46), "Ein"
        Rectangle (583,594 130x46), "Ein"
        Rectangle (736,55 64x370)
        Image (743,55 50x50), image: Icon.P_oben
            OnMouseClick: write the text variable via Default
        Image (743,375 50x50), image: Icon.P_unten
END_VISUALIZATION

// ZY_Visu/Hauptmenu_3/Fusszeile_50
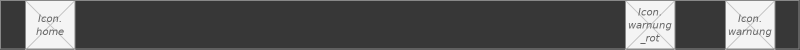
VISUALIZATION Fusszeile_50  // 800x50
    Group (0,0 800x50)
        Rectangle (0,0 800x50)
        Image (625,0 50x50), image: Icon.warnung_rot
            OnMouseClick: execute { Visu.i_Frame_Index:=0; }
        Image (25,0 50x50), image: Icon.home
            OnMouseClick:  Assign=Home_Standard_50, Type=Assignment
            OnMouseClick: execute { Visu.i_Frame_Index:=0; }
        Image (725,0 50x50), image: Icon.warnung
            OnMouseClick:  Assign=Infoseite, Type=Assignment
            OnMouseClick: execute { Visu.i_Frame_Index:=0; }
END_VISUALIZATION

// ZY_Visu/Hauptmenu_3/Hauptmenu
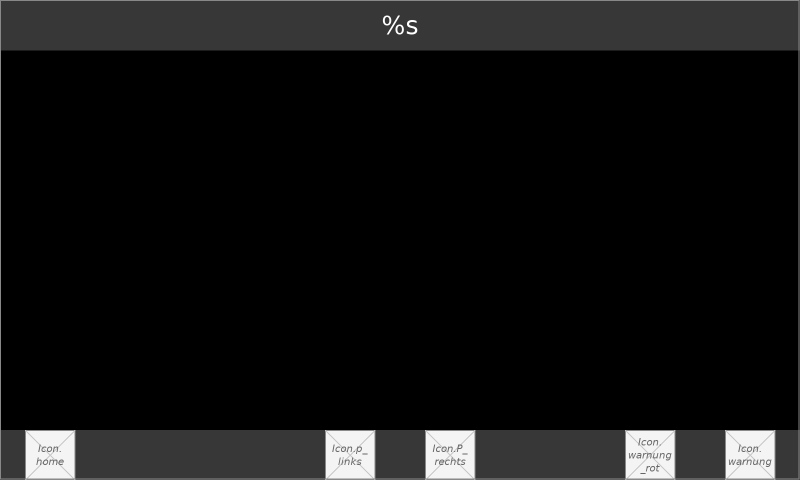
VISUALIZATION Hauptmenu  // 800x480
VAR_IN_OUT
		
END_VAR

VAR
	i_verschieben:INT;

END_VAR
    Image (425,430 50x50), image: Icon.reinnavigieren
    Image (325,430 50x50), image: Icon.reinnavigieren
    Rectangle (0,0 800x50), "%s", text list: 'Sprachen', text index: 32
    Frame (0,430 800x50)
        shows Fusszeile_50()
    Image (425,430 50x50), image: Icon.P_rechts
        OnMouseClick: execute {
            IF i_verschieben>-800 THEN
            	i_verschieben:=i_verschieben-800;
            END_IF
        }
    Image (325,430 50x50), image: Icon.p_links
        OnMouseClick: execute {
            IF i_verschieben<0 THEN
            	i_verschieben:=i_verschieben+800;
            END_IF
        }
    Rectangle (88,515 454x57), "Kachel 1: 0;55 *** Kachel 2: 201;55 *** Kachel 3: 402;55 *** Kachel 4: 604;55 Kachel 5: 0;242 *** Kachel 6: 201;242 *** Kachel 7: 402;242 *** Kachel 8: 604;242"
END_VISUALIZATION

// ZY_Visu/Hauptmenu_3/Kachel_IBN
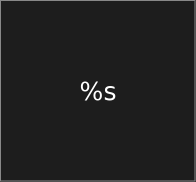
VISUALIZATION Kachel_IBN  // 196x182
    Rectangle (0,0 196x182), "%s", text list: 'Sprachen', text index: 38
END_VISUALIZATION

// ZY_Visu/Hauptmenu_3/Kachel_Konfiguration
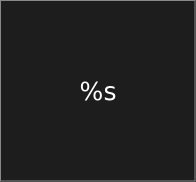
VISUALIZATION Kachel_Konfiguration  // 196x182
    Rectangle (0,0 196x182), "%s", text list: 'Sprachen', text index: 39
END_VISUALIZATION

// ZY_Visu/Hauptmenu_3/Kachel_Kontakt
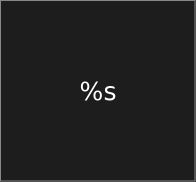
VISUALIZATION Kachel_Kontakt  // 196x182
    Rectangle (0,0 196x182), "%s", text list: 'Sprachen', text index: 40
END_VISUALIZATION

// ZY_Visu/Hauptmenu_3/Kachel_Login
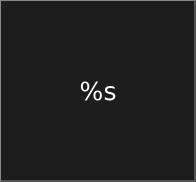
VISUALIZATION Kachel_Login  // 196x182
    Rectangle (0,0 196x182), "%s", text list: 'Sprachen', text index: 34
END_VISUALIZATION

// ZY_Visu/Hauptmenu_3/Kachel_Sollwerte
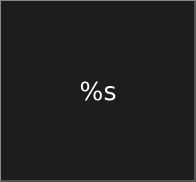
VISUALIZATION Kachel_Sollwerte  // 196x182
    Rectangle (0,0 196x182), "%s", text list: 'Sprachen', text index: 35
END_VISUALIZATION

// ZY_Visu/Hauptmenu_3/Kachel_Sprachen
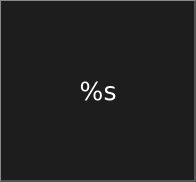
VISUALIZATION Kachel_Sprachen  // 196x182
    Rectangle (0,0 196x182), "%s", text list: 'Sprachen', text index: 33
END_VISUALIZATION

// ZY_Visu/Hauptmenu_3/Kachel_Uhrzeit_einstellen
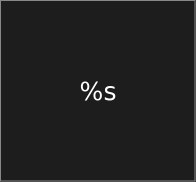
VISUALIZATION Kachel_Uhrzeit_einstellen  // 196x182
    Rectangle (0,0 196x182), "%s", text list: 'Sprachen', text index: 37
END_VISUALIZATION

// ZY_Visu/Hauptmenu_3/Kachel_Verlaufsdiagramm
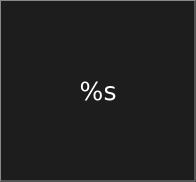
VISUALIZATION Kachel_Verlaufsdiagramm  // 196x182
    Rectangle (0,0 196x182), "%s", text list: 'Sprachen', text index: 36
END_VISUALIZATION

// ZY_Visu/Hauptmenu_3/Kontaktseite
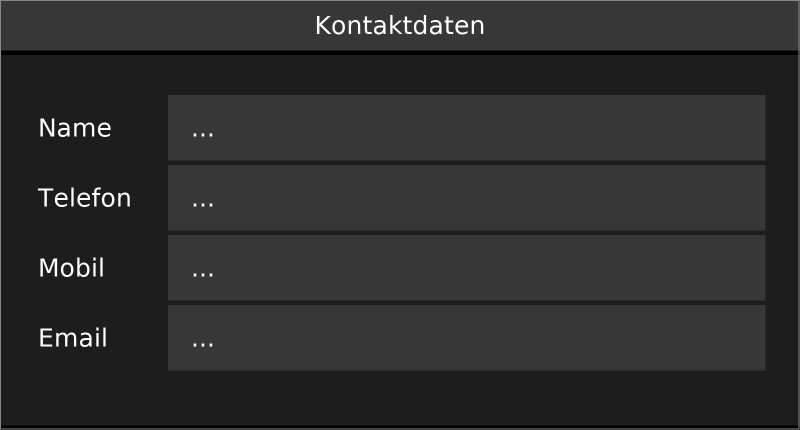
VISUALIZATION Kontaktseite  // 800x430
    Rectangle (0,0 800x50), "Kontaktdaten"
    Rectangle (0,55 800x370)
    Rectangle (168,95 597x65)
    Rectangle (168,165 597x65)
    Rectangle (168,235 597x65)
    Rectangle (168,305 597x65)
    Label (35,95 113x65), "Name"
    Label (35,165 113x65), "Telefon"
    Label (35,235 113x65), "Mobil"
    Label (35,305 113x65), "Email"
    Label (188,305 557x65), "..."
    Label (188,235 557x65), "..."
    Label (188,165 557x65), "..."
    Label (188,95 557x65), "..."
    Frame (0,430 800x50)
        shows Fusszeile_50()
END_VISUALIZATION

// ZY_Visu/Hauptmenu_3/Uhr_einstellen
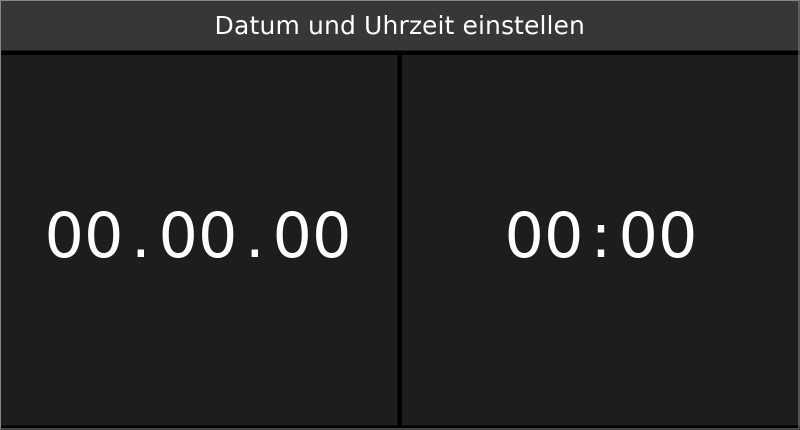
VISUALIZATION Uhr_einstellen  // 800x430
    Frame (0,430 800x50)
        shows Fusszeile_50()
    Rectangle (0,0 800x50), "Datum und Uhrzeit einstellen"
    Rectangle (0,55 397x370)
    Image (425,430 50x50), image: Icon.reinnavigieren
    Image (125,430 50x50), image: Icon.zurueck
        OnMouseClick:  Assign=Hauptmenu, Type=Assignment
    Image (325,430 50x50), image: Icon.reinnavigieren
    Group (402,55 398x370)
        Rectangle (0,0 398x370)
        Group (100,138 198x84)
            Rectangle (84,0 30x84), ":"
            Rectangle (0,0 84x84), "00"
            Rectangle (114,0 84x84), "00"
    Rectangle (156,193 84x84), "00"
    Rectangle (126,193 30x84), "."
    Rectangle (42,193 84x84), "00"
    Rectangle (240,193 30x84), "."
    Rectangle (270,193 84x84), "00"
END_VISUALIZATION

// ZY_Visu/Heizen_Kuehlen/FG_Heizen/FG_Heizen
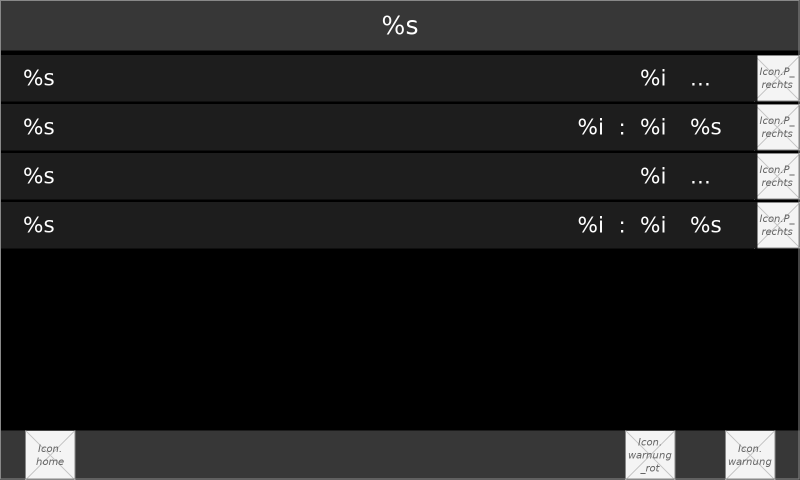
VISUALIZATION FG_Heizen  // 800x480
VAR_IN_OUT
	FB_FG_Heizen:FG_Heizen;
END_VAR
    Frame (0,430 800x50)
        shows Fusszeile_50()
    Frame (0,0 800x430), frame switch variable: GWP_Library.Visu.i_Frame_Index
        shows CLK_W_Wochenprogramm_Liste(i_Titel := 75, FB_CLK_W := FB_CLK_W)
        shows Wochentag_aendern(i_titel := 80, i_Wochentag := FB_CLK_W.t_Ein.wDayOfWeek)
        shows Ein_Aus_Zeit_aendern(i_titel := 68, i_Minuten := FB_CLK_W.t_Ein.wMinute, i_Stunden := FB_CLK_W.t_Ein.wHour)
        shows Wochentag_aendern(i_titel := 80, i_Wochentag := FB_CLK_W.t_Aus.wDayOfWeek)
        shows Ein_Aus_Zeit_aendern(i_titel := 68, i_Minuten := FB_CLK_W.t_Aus.wMinute, i_Stunden := FB_CLK_W.t_Aus.wHour)
END_VISUALIZATION

// ZY_Visu/Heizen_Kuehlen/FG_Heizen/FG_Heizen_Liste
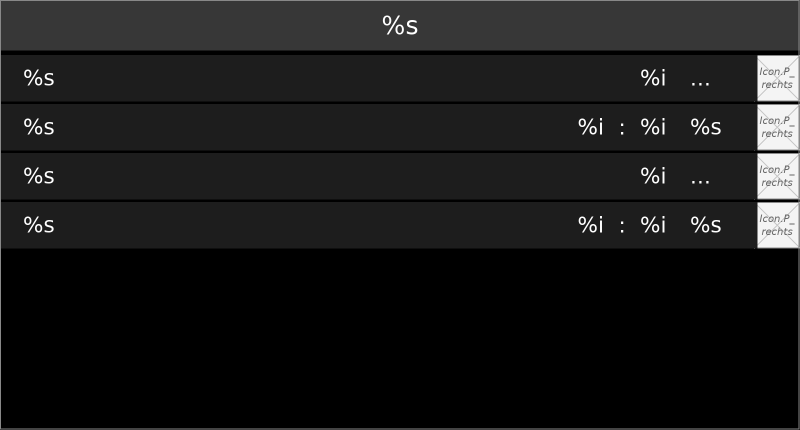
VISUALIZATION FG_Heizen_Liste  // 800x430
VAR_IN_OUT
	FB_FG_Heizen:FG_Heizen;
	
END_VAR
VAR_INPUT
	i_Titel:INT;
END_VAR
	
VAR
	
	
END_VAR
    Rectangle (0,425 800x5)
    Rectangle (0,0 800x50), "%s", text list: 'Sprachen', text index: i_Titel
    Rectangle (0,104 800x46)
    Rectangle (20,104 400x46), "%s", text list: 'Sprachen', text index: 93
    Image (754,104 46x46), image: Icon.P_rechts
        OnMouseClick: execute { Visu.i_Frame_Index:=2; }
    Rectangle (637,104 49x46), "%i", text variable: FB_CLK_W.t_Ein.wMinute
    Rectangle (537,104 70x46), "%i", text variable: FB_CLK_W.t_Ein.wHour
    Rectangle (617,104 10x46), ":"
    Rectangle (687,104 70x46), "%s", text list: 'Sprachen', text index: 74
    Rectangle (0,55 800x46)
    Rectangle (20,55 400x46), "%s", text list: 'Sprachen', text index: 82
    Image (754,55 46x46), image: Icon.P_rechts
        OnMouseClick: execute { Visu.i_Frame_Index:=1; }
    Rectangle (677,55 70x45)
    Rectangle (637,55 49x46), "%i", text variable: FB_CLK_W.t_Ein.wDayOfWeek
    Rectangle (687,55 70x46), "..."
    Rectangle (0,202 800x46)
    Rectangle (20,202 400x46), "%s", text list: 'Sprachen', text index: 94
    Image (754,202 46x46), image: Icon.P_rechts
        OnMouseClick: execute { Visu.i_Frame_Index:=4; }
    Rectangle (637,202 49x46), "%i", text variable: FB_CLK_W.t_Aus.wMinute
    Rectangle (537,202 70x46), "%i", text variable: FB_CLK_W.t_Aus.wHour
    Rectangle (617,202 10x46), ":"
    Rectangle (687,202 70x46), "%s", text list: 'Sprachen', text index: 74
    Rectangle (0,153 800x46)
    Rectangle (20,153 400x46), "%s", text list: 'Sprachen', text index: 83
    Image (754,153 46x46), image: Icon.P_rechts
        OnMouseClick: execute { Visu.i_Frame_Index:=3; }
    Rectangle (677,153 70x45)
    Rectangle (637,153 49x46), "%i", text variable: FB_CLK_W.t_Aus.wDayOfWeek
    Rectangle (687,153 70x46), "..."
END_VISUALIZATION

// ZY_Visu/Heizkurven/Heizkurve
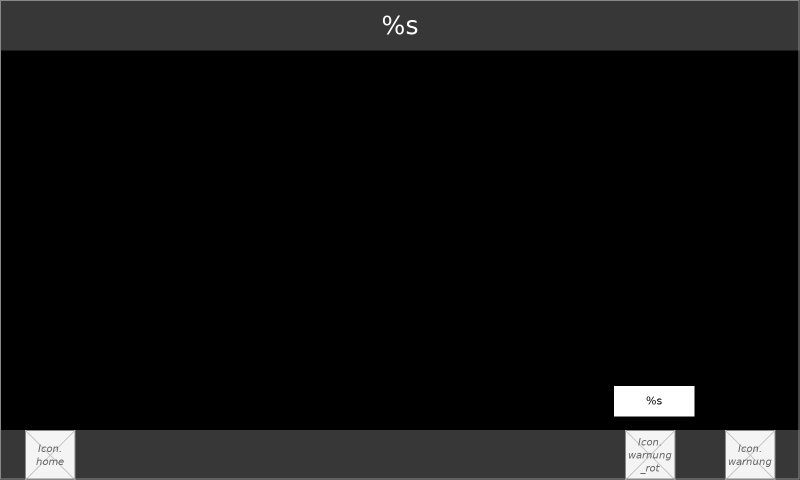
VISUALIZATION Heizkurve  // 800x480
    Image (425,430 50x50), image: Icon.reinnavigieren
    Image (325,430 50x50), image: Icon.reinnavigieren
    Rectangle (0,0 800x50), "%s", text list: 'Sprachen', text index: 71
    Frame (0,430 800x50)
        shows Fusszeile_50()
    Line (154,406)
    Line (143,379) (658,379)
    Line (143,379) (143,90)
    Rectangle (613,385 82x32), "%s"
END_VISUALIZATION

// ZY_Visu/Home/Auswahlmenue
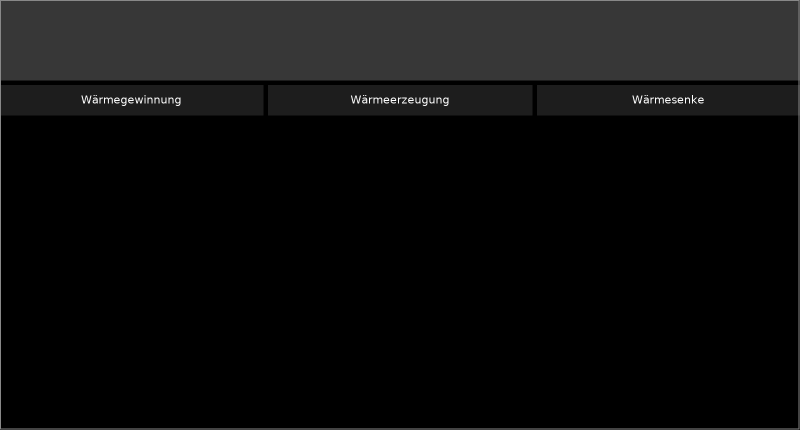
VISUALIZATION Auswahlmenue  // 800x430
    Rectangle (0,0 800x80)
    Rectangle (0,85 263x30), "Wärmegewinnung"
    Rectangle (268,85 264x30), "Wärmeerzeugung"
    Rectangle (537,85 263x30), "Wärmesenke"
END_VISUALIZATION

// ZY_Visu/Home/Ein_Aus_Schalter
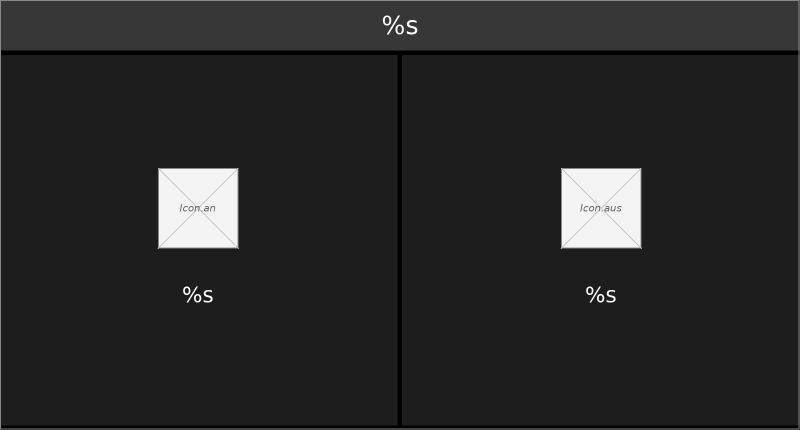
VISUALIZATION Ein_Aus_Schalter  // 800x430
VAR_IN_OUT
		i_Status:INT;
END_VAR

VAR_INPUT
	i_Titel:INT;
	i_Text_1:INT;
	i_Text_2:INT;		
END_VAR

VAR
	x_Aus:BOOL:=TRUE;
	
	
END_VAR
    Rectangle (0,0 800x50), "%s", text list: 'Sprachen', text index: i_Titel
    Group (0,55 397x370)
        OnMouseClick: execute { i_Status:=i_Text_1; }
        Rectangle (0,0 397x370)
        Rectangle (0,0 397x5)
        Image (158,113 80x80), image: Icon.an
        Rectangle (123,225 150x30), "%s", text list: 'Sprachen', text index: i_Text_1
    Image (125,430 50x50), image: Icon.zurueck
        OnMouseClick: execute { Visu.i_Frame_Index:=0; }
    Polygon (943,131)
    Group (402,55 398x370)
        OnMouseClick: execute { i_Status:=i_Text_2; }
        OnMouseClick:  ToggleVariable=x_Aus
        Rectangle (0,0 398x370), colour toggle: x_Aus
        Rectangle (0,0 398x5), colour toggle: x_Aus
        Rectangle (124,225 150x30), "%s", colour toggle: x_Aus, text list: 'Sprachen', text index: i_Text_2
            OnMouseClick: execute {  }
        Image (159,113 80x80), image: Icon.aus
END_VISUALIZATION

// ZY_Visu/Home/Home_Standard_50
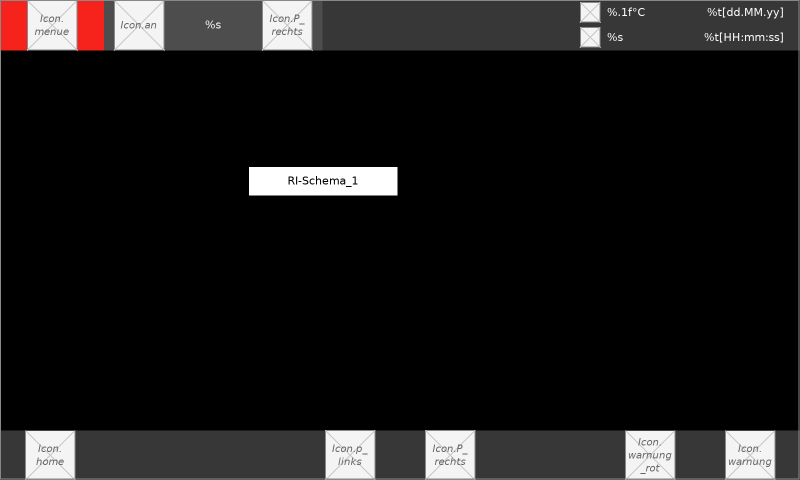
VISUALIZATION Home_Standard_50  // 800x480
VAR_INPUT

END_VAR
	
VAR
	i_Anzeige:INT;	

	

END_VAR
    Frame (0,430 800x50)
        shows Fusszeile_50()
    Frame (0,0 800x430), frame switch variable: Visu.i_Frame_Index
        shows RI_Schema_50(i_Status := i_Anzeige)
        shows Ein_Aus_Schalter(i_Titel := 41, i_Text_1 := 42, i_Text_2 := 43, i_Status := i_Anzeige)
END_VISUALIZATION

// ZY_Visu/Home/RI_Schema_50
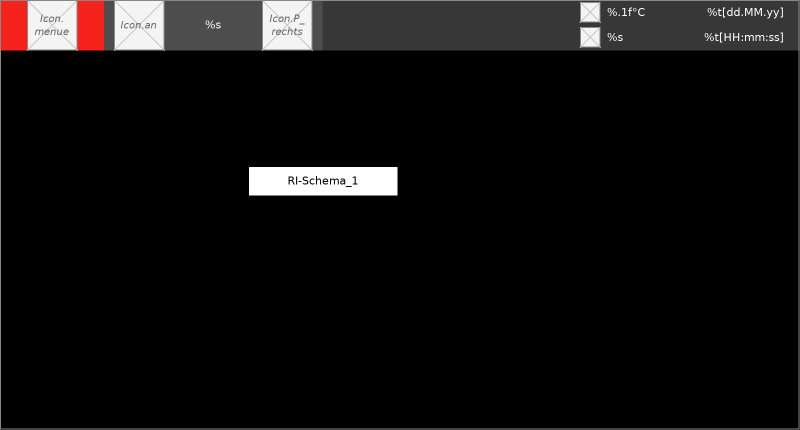
VISUALIZATION RI_Schema_50  // 800x430
VAR
	i_verschieben:INT;
	
END_VAR

VAR_INPUT
	i_Status:INT;

	
	
	
	
END_VAR
    Rectangle (0,0 800x50)
    Rectangle (702,0 85x25), "%t[dd.MM.yy]"
    Rectangle (702,25 85x25), "%t[HH:mm:ss]"
    Image (580,27 20x20), image: Icon.login_status
    Rectangle (604,0 85x25), "%.1f°C"
    Rectangle (604,25 85x25), "%s"
    Group (0,0 104x50)
        OnMouseClick:  Assign=Hauptmenu, Type=Assignment
        Rectangle (0,0 104x50)
        Image (27,0 50x50), image: Icon.menue
    Image (425,430 50x50), image: Icon.P_rechts
        OnMouseClick: execute {
            IF i_verschieben>-800 THEN
            	i_verschieben:=i_verschieben-400;
            END_IF
        }
    Image (325,430 50x50), image: Icon.p_links
        OnMouseClick: execute {
            IF i_verschieben<0 THEN
            	i_verschieben:=i_verschieben+400;
            END_IF
        }
    Image (580,2 20x20), image: Icon.aussentemperatur
    Rectangle (104,0 218x50), "%s", text list: 'Sprachen', text index: i_Status
    Image (114,0 50x50), image: Icon.an
    Image (262,0 50x50), image: Icon.P_rechts
        OnMouseClick: execute { Visu.i_Frame_Index:=1; }
    Group (248,166 842x88)
        p3560616238: i_verschieben
        Rectangle (0,0 150x30), "RI-Schema_1"
        Rectangle (698,58 150x30), "RI-Schema_2"
END_VISUALIZATION

// ZY_Visu/IBN/IO_Auswahl
